LIN {X 0,Y 420.571,Z 343.007,A -85,B 0,C 180,E1 -10184.764,E2 -10184.764} C_VEL
LIN {X 0,Y 421.364,Z 331.747,A -85,B 0,C 180,E1 -10185.601,E2 -10185.601} C_VEL
LIN {X 0,Y 422.031,Z 320.369,A -85,B 0,C 180,E1 -10186.258,E2 -10186.258} C_VEL
LIN {X 0,Y 422.669,Z 307.508,A -85,B 0,C 180,E1 -10186.792,E2 -10186.792} C_VEL
LIN {X 0,Y 423.083,Z 294.135,A -85,B 0,C 180,E1 -10187.148,E2 -10187.148} C_VEL
LIN {X 0,Y 424.009,Z 215.37,A -85,B 0,C 180,E1 -10188.601,E2 -10188.601} C_VEL
LIN {X 0,Y 420.22,Z 192.517,A -85,B 0,C 180,E1 -10189.238,E2 -10189.238} C_VEL
LIN {X 0,Y 419.835,Z 190.333,A -85,B 0,C 180,E1 -10189.315,E2 -10189.315} C_VEL
LIN {X 0,Y 420.887,Z 173.807,A -85,B 0,C 180,E1 -10192.585,E2 -10192.585} C_VEL
LIN {X 0,Y 421.24,Z 166.164,A -85,B 0,C 180,E1 -10194.126,E2 -10194.126} C_VEL
LIN {X 0,Y 418.93,Z 154.675,A -85,B 0,C 180,E1 -10196.664,E2 -10196.664} C_VEL
LIN {X 0,Y 418.192,Z 151.4,A -85,B 0,C 180,E1 -10197.451,E2 -10197.451} C_VEL
LIN {X 0,Y 418.233,Z 151.395,A -85,B 0,C 180,E1 -10200.272,E2 -10200.272} C_VEL
LIN {X 0,Y 418.229,Z 151.389,A -85,B 0,C 180,E1 -10203.678,E2 -10203.678} C_VEL
LIN {X 0,Y 418.231,Z 151.392,A -85,B 0,C 180,E1 -10207.224,E2 -10207.224} C_VEL
LIN {X 0,Y 418.204,Z 151.395,A -85,B 0,C 180,E1 -10210.866,E2 -10210.866} C_VEL
LIN {X 0,Y 418.199,Z 151.393,A -85,B 0,C 180,E1 -10213.727,E2 -10213.727} C_VEL
LIN {X 0,Y 418.195,Z 151.394,A -85,B 0,C 180,E1 -10216.446,E2 -10216.446} C_VEL
LIN {X 0,Y 418.203,Z 151.392,A -85,B 0,C 180,E1 -10219.132,E2 -10219.132} C_VEL
LIN {X 0,Y 418.229,Z 151.388,A -85,B 0,C 180,E1 -10222.774,E2 -10222.774} C_VEL
LIN {X 0,Y 418.226,Z 151.387,A -85,B 0,C 180,E1 -10226.32,E2 -10226.32} C_VEL
LIN {X 0,Y 418.228,Z 151.383,A -85,B 0,C 180,E1 -10229.726,E2 -10229.726} C_VEL
LIN {X 0,Y 418.202,Z 151.386,A -85,B 0,C 180,E1 -10233.016,E2 -10233.016} C_VEL
LIN {X 0,Y 418.248,Z 151.388,A -85,B 0,C 180,E1 -10236.216,E2 -10236.216} C_VEL
LIN {X 0,Y 418.229,Z 151.386,A -85,B 0,C 180,E1 -10239.336,E2 -10239.336} C_VEL
LIN {X 0,Y 418.23,Z 151.389,A -85,B 0,C 180,E1 -10242.393,E2 -10242.393} C_VEL
LIN {X 0,Y 418.268,Z 151.378,A -85,B 0,C 180,E1 -10245.401,E2 -10245.401} C_VEL
LIN {X 0,Y 418.295,Z 151.377,A -85,B 0,C 180,E1 -10248.368,E2 -10248.368} C_VEL
LIN {X 0,Y 418.439,Z 151.361,A -85,B 0,C 180,E1 -10252.278,E2 -10252.278} C_VEL
LIN {X 0,Y 418.461,Z 151.358,A -85,B 0,C 180,E1 -10254.216,E2 -10254.216} C_VEL
LIN {X 0,Y 418.525,Z 151.351,A -85,B 0,C 180,E1 -10258.075,E2 -10258.075} C_VEL
LIN {X 0,Y 418.398,Z 151.362,A -85,B 0,C 180,E1 -10260.962,E2 -10260.962} C_VEL
LIN {X 0,Y 418.46,Z 151.357,A -85,B 0,C 180,E1 -10262.888,E2 -10262.888} C_VEL
LIN {X 0,Y 418.432,Z 151.362,A -85,B 0,C 180,E1 -10266.752,E2 -10266.752} C_VEL
LIN {X 0,Y 418.313,Z 151.381,A -85,B 0,C 180,E1 -10269.672,E2 -10269.672} C_VEL
LIN {X 0,Y 418.338,Z 151.379,A -85,B 0,C 180,E1 -10273,E2 -10273} C_VEL
LIN {X 0,Y 418.251,Z 151.388,A -85,B 0,C 180,E1 -10276.71,E2 -10276.71} C_VEL
LIN {X 0,Y 418.259,Z 151.388,A -85,B 0,C 180,E1 -10280.165,E2 -10280.165} C_VEL
LIN {X 0,Y 418.281,Z 151.439,A -85,B 0,C 180,E1 -10280.537,E2 -10280.537} C_VEL
LIN {X 0,Y 420.491,Z 162.689,A -85,B 0,C 180,E1 -10283.184,E2 -10283.184} C_VEL
LIN {X 0,Y 420.261,Z 170.089,A -85,B 0,C 180,E1 -10284.776,E2 -10284.776} C_VEL
LIN {X 0,Y 424.452,Z 189.753,A -85,B 0,C 180,E1 -10285.38,E2 -10285.38} C_VEL
LIN {X 0,Y 423.071,Z 278.399,A -85,B 0,C 180,E1 -10287.032,E2 -10287.032} C_VEL
LIN {X 0,Y 422.599,Z 291.851,A -85,B 0,C 180,E1 -10287.483,E2 -10287.483} C_VEL
LIN {X 0,Y 422.146,Z 303.797,A -85,B 0,C 180,E1 -10288.074,E2 -10288.074} C_VEL
LIN {X 0,Y 421.53,Z 314.904,A -85,B 0,C 180,E1 -10288.802,E2 -10288.802} C_VEL
LIN {X 0,Y 420.809,Z 325.924,A -85,B 0,C 180,E1 -10289.722,E2 -10289.722} C_VEL
LIN {X 0,Y 420.053,Z 336.491,A -85,B 0,C 180,E1 -10290.823,E2 -10290.823} C_VEL
LIN {X 0,Y 419.339,Z 345.705,A -85,B 0,C 180,E1 -10292.006,E2 -10292.006} C_VEL
LIN {X 0,Y 418.597,Z 354.791,A -85,B 0,C 180,E1 -10293.46,E2 -10293.46} C_VEL
LIN {X 0,Y 418.121,Z 361.803,A -85,B 0,C 180,E1 -10294.854,E2 -10294.854} C_VEL
LIN {X 0,Y 417.75,Z 367.093,A -85,B 0,C 180,E1 -10296.147,E2 -10296.147} C_VEL
LIN {X 0,Y 417.463,Z 372.148,A -85,B 0,C 180,E1 -10297.699,E2 -10297.699} C_VEL
LIN {X 0,Y 417.19,Z 375.839,A -85,B 0,C 180,E1 -10299.204,E2 -10299.204} C_VEL
LIN {X 0,Y 416.986,Z 378.927,A -85,B 0,C 180,E1 -10301.095,E2 -10301.095} C_VEL
LIN {X 0,Y 416.87,Z 380.157,A -85,B 0,C 180,E1 -10302.404,E2 -10302.404} C_VEL
LIN {X 0,Y 416.855,Z 380.606,A -85,B 0,C 180,E1 -10303.728,E2 -10303.728} C_VEL
LIN {X 0,Y 416.898,Z 380.294,A -85,B 0,C 180,E1 -10305.074,E2 -10305.074} C_VEL
LIN {X 0,Y 416.93,Z 379.175,A -85,B 0,C 180,E1 -10306.454,E2 -10306.454} C_VEL
LIN {X 0,Y 417.024,Z 377.173,A -85,B 0,C 180,E1 -10307.86,E2 -10307.86} C_VEL
LIN {X 0,Y 417.209,Z 374.191,A -85,B 0,C 180,E1 -10309.291,E2 -10309.291} C_VEL
LIN {X 0,Y 417.417,Z 370.056,A -85,B 0,C 180,E1 -10310.759,E2 -10310.759} C_VEL
LIN {X 0,Y 417.738,Z 364.602,A -85,B 0,C 180,E1 -10312.253,E2 -10312.253} C_VEL
LIN {X 0,Y 418.142,Z 357.548,A -85,B 0,C 180,E1 -10313.781,E2 -10313.781} C_VEL
LIN {X 0,Y 418.699,Z 349.368,A -85,B 0,C 180,E1 -10315.202,E2 -10315.202} C_VEL
LIN {X 0,Y 419.339,Z 340.676,A -85,B 0,C 180,E1 -10316.423,E2 -10316.423} C_VEL
LIN {X 0,Y 420.009,Z 330.101,A -85,B 0,C 180,E1 -10317.626,E2 -10317.626} C_VEL
LIN {X 0,Y 420.68,Z 318.982,A -85,B 0,C 180,E1 -10318.64,E2 -10318.64} C_VEL
LIN {X 0,Y 421.334,Z 307.001,A -85,B 0,C 180,E1 -10319.489,E2 -10319.489} C_VEL
LIN {X 0,Y 421.864,Z 294.615,A -85,B 0,C 180,E1 -10320.153,E2 -10320.153} C_VEL
LIN {X 0,Y 422.251,Z 281.602,A -85,B 0,C 180,E1 -10320.646,E2 -10320.646} C_VEL
LIN {X 0,Y 422.49,Z 266.058,A -85,B 0,C 180,E1 -10320.988,E2 -10320.988} C_VEL
LIN {X 0,Y 423.528,Z 189.194,A -85,B 0,C 180,E1 -10322.371,E2 -10322.371} C_VEL
LIN {X 0,Y 419.842,Z 169.494,A -85,B 0,C 180,E1 -10322.926,E2 -10322.926} C_VEL
LIN {X 0,Y 420.197,Z 162.178,A -85,B 0,C 180,E1 -10324.578,E2 -10324.578} C_VEL
LIN {X 0,Y 419.152,Z 156.176,A -85,B 0,C 180,E1 -10326.018,E2 -10326.018} C_VEL
LIN {X 0,Y 418.154,Z 154.508,A -85,B 0,C 180,E1 -10326.497,E2 -10326.497} C_VEL
LIN {X 0,Y 416.324,Z 153.399,A -85,B 0,C 180,E1 -10326.973,E2 -10326.973} C_VEL
LIN {X 0,Y 412.363,Z 152.396,A -85,B 0,C 180,E1 -10327.956,E2 -10327.956} C_VEL
LIN {X 0,Y 411.2,Z 152.268,A -85,B 0,C 180,E1 -10328.589,E2 -10328.589} C_VEL
LIN {X 0,Y 411.179,Z 152.266,A -85,B 0,C 180,E1 -10328.683,E2 -10328.683} C_VEL
LIN {X 0,Y 411.209,Z 152.262,A -85,B 0,C 180,E1 -10332.083,E2 -10332.083} C_VEL
LIN {X 0,Y 411.227,Z 152.257,A -85,B 0,C 180,E1 -10335.147,E2 -10335.147} C_VEL
LIN {X 0,Y 411.27,Z 152.256,A -85,B 0,C 180,E1 -10338.167,E2 -10338.167} C_VEL
LIN {X 0,Y 411.384,Z 152.243,A -85,B 0,C 180,E1 -10342.145,E2 -10342.145} C_VEL
LIN {X 0,Y 411.424,Z 152.238,A -85,B 0,C 180,E1 -10344.118,E2 -10344.118} C_VEL
LIN {X 0,Y 411.498,Z 152.229,A -85,B 0,C 180,E1 -10348.043,E2 -10348.043} C_VEL
LIN {X 0,Y 411.373,Z 152.239,A -85,B 0,C 180,E1 -10350.979,E2 -10350.979} C_VEL
LIN {X 0,Y 411.423,Z 152.232,A -85,B 0,C 180,E1 -10352.938,E2 -10352.938} C_VEL
LIN {X 0,Y 411.386,Z 152.237,A -85,B 0,C 180,E1 -10356.868,E2 -10356.868} C_VEL
LIN {X 0,Y 411.272,Z 152.258,A -85,B 0,C 180,E1 -10359.839,E2 -10359.839} C_VEL
LIN {X 0,Y 411.302,Z 152.248,A -85,B 0,C 180,E1 -10363.103,E2 -10363.103} C_VEL
LIN {X 0,Y 411.203,Z 152.26,A -85,B 0,C 180,E1 -10366.891,E2 -10366.891} C_VEL
LIN {X 0,Y 411.2,Z 152.263,A -85,B 0,C 180,E1 -10369.988,E2 -10369.988} C_VEL
LIN {X 0,Y 411.182,Z 152.265,A -85,B 0,C 180,E1 -10373.149,E2 -10373.149} C_VEL
LIN {X 0,Y 411.166,Z 152.264,A -85,B 0,C 180,E1 -10376.386,E2 -10376.386} C_VEL
LIN {X 0,Y 411.188,Z 152.265,A -85,B 0,C 180,E1 -10379.713,E2 -10379.713} C_VEL
LIN {X 0,Y 411.199,Z 152.265,A -85,B 0,C 180,E1 -10383.156,E2 -10383.156} C_VEL
LIN {X 0,Y 411.186,Z 152.262,A -85,B 0,C 180,E1 -10386.552,E2 -10386.552} C_VEL
LIN {X 0,Y 411.163,Z 152.266,A -85,B 0,C 180,E1 -10389.72,E2 -10389.72} C_VEL
LIN {X 0,Y 411.157,Z 152.273,A -85,B 0,C 180,E1 -10393.135,E2 -10393.135} C_VEL
LIN {X 0,Y 411.158,Z 152.266,A -85,B 0,C 180,E1 -10395.882,E2 -10395.882} C_VEL
LIN {X 0,Y 411.152,Z 152.268,A -85,B 0,C 180,E1 -10399.493,E2 -10399.493} C_VEL
LIN {X 0,Y 411.175,Z 152.263,A -85,B 0,C 180,E1 -10402.025,E2 -10402.025} C_VEL
LIN {X 0,Y 411.195,Z 152.265,A -85,B 0,C 180,E1 -10405.124,E2 -10405.124} C_VEL
LIN {X 0,Y 411.157,Z 152.266,A -85,B 0,C 180,E1 -10408.003,E2 -10408.003} C_VEL
LIN {X 0,Y 411.165,Z 152.265,A -85,B 0,C 180,E1 -10411.406,E2 -10411.406} C_VEL
LIN {X 0,Y 411.182,Z 152.266,A -85,B 0,C 180,E1 -10414.941,E2 -10414.941} C_VEL
LIN {X 0,Y 411.194,Z 152.262,A -85,B 0,C 180,E1 -10417.913,E2 -10417.913} C_VEL
LIN {X 0,Y 411.208,Z 152.261,A -85,B 0,C 180,E1 -10421.051,E2 -10421.051} C_VEL
LIN {X 0,Y 411.205,Z 152.263,A -85,B 0,C 180,E1 -10424.13,E2 -10424.13} C_VEL
LIN {X 0,Y 411.296,Z 152.248,A -85,B 0,C 180,E1 -10427.166,E2 -10427.166} C_VEL
LIN {X 0,Y 411.268,Z 152.257,A -85,B 0,C 180,E1 -10430.161,E2 -10430.161} C_VEL
LIN {X 0,Y 411.384,Z 152.237,A -85,B 0,C 180,E1 -10433.132,E2 -10433.132} C_VEL
LIN {X 0,Y 411.278,Z 152.25,A -85,B 0,C 180,E1 -10435.099,E2 -10435.099} C_VEL
LIN {X 0,Y 411.496,Z 152.23,A -85,B 0,C 180,E1 -10438.043,E2 -10438.043} C_VEL
LIN {X 0,Y 411.371,Z 152.239,A -85,B 0,C 180,E1 -10440.979,E2 -10440.979} C_VEL
LIN {X 0,Y 411.42,Z 152.233,A -85,B 0,C 180,E1 -10442.938,E2 -10442.938} C_VEL
LIN {X 0,Y 411.384,Z 152.237,A -85,B 0,C 180,E1 -10446.869,E2 -10446.869} C_VEL
LIN {X 0,Y 411.27,Z 152.259,A -85,B 0,C 180,E1 -10449.84,E2 -10449.84} C_VEL
LIN {X 0,Y 411.301,Z 152.248,A -85,B 0,C 180,E1 -10453.104,E2 -10453.104} C_VEL
LIN {X 0,Y 411.203,Z 152.26,A -85,B 0,C 180,E1 -10456.891,E2 -10456.891} C_VEL
LIN {X 0,Y 411.2,Z 152.263,A -85,B 0,C 180,E1 -10459.989,E2 -10459.989} C_VEL
LIN {X 0,Y 411.182,Z 152.265,A -85,B 0,C 180,E1 -10463.149,E2 -10463.149} C_VEL
LIN {X 0,Y 411.167,Z 152.264,A -85,B 0,C 180,E1 -10466.386,E2 -10466.386} C_VEL
LIN {X 0,Y 411.189,Z 152.265,A -85,B 0,C 180,E1 -10469.714,E2 -10469.714} C_VEL
LIN {X 0,Y 411.201,Z 152.265,A -85,B 0,C 180,E1 -10473.157,E2 -10473.157} C_VEL
LIN {X 0,Y 411.186,Z 152.263,A -85,B 0,C 180,E1 -10476.552,E2 -10476.552} C_VEL
LIN {X 0,Y 411.166,Z 152.266,A -85,B 0,C 180,E1 -10479.721,E2 -10479.721} C_VEL
LIN {X 0,Y 411.159,Z 152.272,A -85,B 0,C 180,E1 -10483.136,E2 -10483.136} C_VEL
LIN {X 0,Y 411.162,Z 152.265,A -85,B 0,C 180,E1 -10485.882,E2 -10485.882} C_VEL
LIN {X 0,Y 411.157,Z 152.267,A -85,B 0,C 180,E1 -10489.493,E2 -10489.493} C_VEL
LIN {X 0,Y 411.18,Z 152.263,A -85,B 0,C 180,E1 -10492.025,E2 -10492.025} C_VEL
LIN {X 0,Y 411.201,Z 152.264,A -85,B 0,C 180,E1 -10495.124,E2 -10495.124} C_VEL
LIN {X 0,Y 411.158,Z 152.266,A -85,B 0,C 180,E1 -10498.002,E2 -10498.002} C_VEL
LIN {X 0,Y 411.169,Z 152.267,A -85,B 0,C 180,E1 -10501.407,E2 -10501.407} C_VEL
LIN {X 0,Y 411.198,Z 152.412,A -85,B 0,C 180,E1 -10502.635,E2 -10502.635} C_VEL
LIN {X 0,Y 413.704,Z 164.762,A -85,B 0,C 180,E1 -10505.405,E2 -10505.405} C_VEL
LIN {X 0,Y 414.113,Z 168.81,A -85,B 0,C 180,E1 -10506.273,E2 -10506.273} C_VEL
LIN {X 0,Y 412.889,Z 187.598,A -85,B 0,C 180,E1 -10510.097,E2 -10510.097} C_VEL
LIN {X 0,Y 412.57,Z 191.176,A -85,B 0,C 180,E1 -10510.815,E2 -10510.815} C_VEL
LIN {X 0,Y 416.564,Z 216.973,A -85,B 0,C 180,E1 -10511.482,E2 -10511.482} C_VEL
LIN {X 0,Y 415.425,Z 299,A -85,B 0,C 180,E1 -10513.001,E2 -10513.001} C_VEL
LIN {X 0,Y 414.972,Z 312.17,A -85,B 0,C 180,E1 -10513.425,E2 -10513.425} C_VEL
LIN {X 0,Y 414.389,Z 324.339,A -85,B 0,C 180,E1 -10514.002,E2 -10514.002} C_VEL
LIN {X 0,Y 413.724,Z 335.853,A -85,B 0,C 180,E1 -10514.734,E2 -10514.734} C_VEL
LIN {X 0,Y 413.008,Z 346.776,A -85,B 0,C 180,E1 -10515.627,E2 -10515.627} C_VEL
LIN {X 0,Y 412.258,Z 358.362,A -85,B 0,C 180,E1 -10516.826,E2 -10516.826} C_VEL
LIN {X 0,Y 411.689,Z 366.989,A -85,B 0,C 180,E1 -10517.929,E2 -10517.929} C_VEL
LIN {X 0,Y 411.068,Z 374.981,A -85,B 0,C 180,E1 -10519.16,E2 -10519.16} C_VEL
LIN {X 0,Y 410.605,Z 382.783,A -85,B 0,C 180,E1 -10520.642,E2 -10520.642} C_VEL
LIN {X 0,Y 410.285,Z 389.031,A -85,B 0,C 180,E1 -10522.124,E2 -10522.124} C_VEL
LIN {X 0,Y 410.071,Z 394.382,A -85,B 0,C 180,E1 -10523.741,E2 -10523.741} C_VEL
LIN {X 0,Y 410.016,Z 397.784,A -85,B 0,C 180,E1 -10525.083,E2 -10525.083} C_VEL
LIN {X 0,Y 409.932,Z 399.737,A -85,B 0,C 180,E1 -10526.068,E2 -10526.068} C_VEL
LIN {X 0,Y 409.927,Z 401.26,A -85,B 0,C 180,E1 -10527.052,E2 -10527.052} C_VEL
LIN {X 0,Y 409.967,Z 402.321,A -85,B 0,C 180,E1 -10528.035,E2 -10528.035} C_VEL
LIN {X 0,Y 409.937,Z 402.979,A -85,B 0,C 180,E1 -10529.018,E2 -10529.018} C_VEL
LIN {X 0,Y 409.928,Z 403.244,A -85,B 0,C 180,E1 -10530,E2 -10530} C_VEL
LIN {X 0,Y 409.937,Z 403.101,A -85,B 0,C 180,E1 -10530.982,E2 -10530.982} C_VEL
LIN {X 0,Y 409.967,Z 402.517,A -85,B 0,C 180,E1 -10531.965,E2 -10531.965} C_VEL
LIN {X 0,Y 409.925,Z 401.535,A -85,B 0,C 180,E1 -10532.948,E2 -10532.948} C_VEL
LIN {X 0,Y 409.931,Z 400.152,A -85,B 0,C 180,E1 -10533.932,E2 -10533.932} C_VEL
LIN {X 0,Y 410.012,Z 397.234,A -85,B 0,C 180,E1 -10535.409,E2 -10535.409} C_VEL
LIN {X 0,Y 410.168,Z 393.27,A -85,B 0,C 180,E1 -10536.888,E2 -10536.888} C_VEL
LIN {X 0,Y 410.475,Z 387.186,A -85,B 0,C 180,E1 -10538.616,E2 -10538.616} C_VEL
LIN {X 0,Y 410.914,Z 380.501,A -85,B 0,C 180,E1 -10540.096,E2 -10540.096} C_VEL
LIN {X 0,Y 411.512,Z 372.217,A -85,B 0,C 180,E1 -10541.576,E2 -10541.576} C_VEL
LIN {X 0,Y 412.276,Z 363.768,A -85,B 0,C 180,E1 -10542.803,E2 -10542.803} C_VEL
LIN {X 0,Y 412.884,Z 354.377,A -85,B 0,C 180,E1 -10543.93,E2 -10543.93} C_VEL
LIN {X 0,Y 413.697,Z 343.103,A -85,B 0,C 180,E1 -10545.015,E2 -10545.015} C_VEL
LIN {X 0,Y 414.549,Z 331.915,A -85,B 0,C 180,E1 -10545.865,E2 -10545.865} C_VEL
LIN {X 0,Y 415.239,Z 320.652,A -85,B 0,C 180,E1 -10546.532,E2 -10546.532} C_VEL
LIN {X 0,Y 415.858,Z 308.078,A -85,B 0,C 180,E1 -10547.075,E2 -10547.075} C_VEL
LIN {X 0,Y 416.322,Z 295.194,A -85,B 0,C 180,E1 -10547.436,E2 -10547.436} C_VEL
LIN {X 0,Y 417.379,Z 216.328,A -85,B 0,C 180,E1 -10548.919,E2 -10548.919} C_VEL
LIN {X 0,Y 413.666,Z 194.049,A -85,B 0,C 180,E1 -10549.561,E2 -10549.561} C_VEL
LIN {X 0,Y 412.977,Z 190.144,A -85,B 0,C 180,E1 -10549.685,E2 -10549.685} C_VEL
LIN {X 0,Y 414.183,Z 172.189,A -85,B 0,C 180,E1 -10553.309,E2 -10553.309} C_VEL
LIN {X 0,Y 414.313,Z 167.438,A -85,B 0,C 180,E1 -10554.289,E2 -10554.289} C_VEL
LIN {X 0,Y 411.997,Z 156.051,A -85,B 0,C 180,E1 -10556.865,E2 -10556.865} C_VEL
LIN {X 0,Y 411.173,Z 152.274,A -85,B 0,C 180,E1 -10557.76,E2 -10557.76} C_VEL
LIN {X 0,Y 411.182,Z 152.274,A -85,B 0,C 180,E1 -10560.848,E2 -10560.848} C_VEL
LIN {X 0,Y 411.19,Z 152.265,A -85,B 0,C 180,E1 -10564.334,E2 -10564.334} C_VEL
LIN {X 0,Y 411.183,Z 152.268,A -85,B 0,C 180,E1 -10566.742,E2 -10566.742} C_VEL
LIN {X 0,Y 411.165,Z 152.27,A -85,B 0,C 180,E1 -10569.719,E2 -10569.719} C_VEL
LIN {X 0,Y 411.159,Z 152.273,A -85,B 0,C 180,E1 -10573.134,E2 -10573.134} C_VEL
LIN {X 0,Y 411.159,Z 152.268,A -85,B 0,C 180,E1 -10575.881,E2 -10575.881} C_VEL
LIN {X 0,Y 411.154,Z 152.267,A -85,B 0,C 180,E1 -10579.492,E2 -10579.492} C_VEL
LIN {X 0,Y 411.177,Z 152.265,A -85,B 0,C 180,E1 -10582.024,E2 -10582.024} C_VEL
LIN {X 0,Y 411.197,Z 152.264,A -85,B 0,C 180,E1 -10585.123,E2 -10585.123} C_VEL
LIN {X 0,Y 411.154,Z 152.267,A -85,B 0,C 180,E1 -10588.001,E2 -10588.001} C_VEL
LIN {X 0,Y 411.163,Z 152.266,A -85,B 0,C 180,E1 -10591.405,E2 -10591.405} C_VEL
LIN {X 0,Y 411.182,Z 152.266,A -85,B 0,C 180,E1 -10594.941,E2 -10594.941} C_VEL
LIN {X 0,Y 411.192,Z 152.258,A -85,B 0,C 180,E1 -10597.912,E2 -10597.912} C_VEL
LIN {X 0,Y 411.176,Z 152.26,A -85,B 0,C 180,E1 -10601.049,E2 -10601.049} C_VEL
LIN {X 0,Y 411.201,Z 152.263,A -85,B 0,C 180,E1 -10604.129,E2 -10604.129} C_VEL
LIN {X 0,Y 411.295,Z 152.249,A -85,B 0,C 180,E1 -10607.165,E2 -10607.165} C_VEL
LIN {X 0,Y 411.268,Z 152.259,A -85,B 0,C 180,E1 -10610.16,E2 -10610.16} C_VEL
LIN {X 0,Y 411.382,Z 152.239,A -85,B 0,C 180,E1 -10613.131,E2 -10613.131} C_VEL
LIN {X 0,Y 411.276,Z 152.248,A -85,B 0,C 180,E1 -10615.098,E2 -10615.098} C_VEL
LIN {X 0,Y 411.494,Z 152.227,A -85,B 0,C 180,E1 -10618.042,E2 -10618.042} C_VEL
LIN {X 0,Y 411.368,Z 152.238,A -85,B 0,C 180,E1 -10620.978,E2 -10620.978} C_VEL
LIN {X 0,Y 411.419,Z 152.235,A -85,B 0,C 180,E1 -10622.937,E2 -10622.937} C_VEL
LIN {X 0,Y 411.382,Z 152.24,A -85,B 0,C 180,E1 -10626.868,E2 -10626.868} C_VEL
LIN {X 0,Y 411.267,Z 152.26,A -85,B 0,C 180,E1 -10629.839,E2 -10629.839} C_VEL
LIN {X 0,Y 411.297,Z 152.257,A -85,B 0,C 180,E1 -10633.103,E2 -10633.103} C_VEL
LIN {X 0,Y 411.2,Z 152.267,A -85,B 0,C 180,E1 -10636.891,E2 -10636.891} C_VEL
LIN {X 0,Y 411.234,Z 152.347,A -85,B 0,C 180,E1 -10640.214,E2 -10640.214} C_VEL
LIN {X 0,Y 413.559,Z 163.936,A -85,B 0,C 180,E1 -10643.008,E2 -10643.008} C_VEL
LIN {X 0,Y 413.416,Z 170.133,A -85,B 0,C 180,E1 -10644.379,E2 -10644.379} C_VEL
LIN {X 0,Y 417.825,Z 190.845,A -85,B 0,C 180,E1 -10645.057,E2 -10645.057} C_VEL
LIN {X 0,Y 416.347,Z 278.62,A -85,B 0,C 180,E1 -10646.721,E2 -10646.721} C_VEL
LIN {X 0,Y 415.857,Z 292.111,A -85,B 0,C 180,E1 -10647.182,E2 -10647.182} C_VEL
LIN {X 0,Y 415.375,Z 304.284,A -85,B 0,C 180,E1 -10647.797,E2 -10647.797} C_VEL
LIN {X 0,Y 414.637,Z 316.272,A -85,B 0,C 180,E1 -10648.609,E2 -10648.609} C_VEL
LIN {X 0,Y 413.835,Z 327.728,A -85,B 0,C 180,E1 -10649.605,E2 -10649.605} C_VEL
LIN {X 0,Y 413.103,Z 337.69,A -85,B 0,C 180,E1 -10650.689,E2 -10650.689} C_VEL
LIN {X 0,Y 412.349,Z 346.691,A -85,B 0,C 180,E1 -10651.894,E2 -10651.894} C_VEL
LIN {X 0,Y 411.561,Z 355.998,A -85,B 0,C 180,E1 -10653.44,E2 -10653.44} C_VEL
LIN {X 0,Y 411.062,Z 362.796,A -85,B 0,C 180,E1 -10654.85,E2 -10654.85} C_VEL
LIN {X 0,Y 410.606,Z 368.893,A -85,B 0,C 180,E1 -10656.443,E2 -10656.443} C_VEL
LIN {X 0,Y 410.3,Z 373.675,A -85,B 0,C 180,E1 -10658.071,E2 -10658.071} C_VEL
LIN {X 0,Y 410.05,Z 376.872,A -85,B 0,C 180,E1 -10659.533,E2 -10659.533} C_VEL
LIN {X 0,Y 409.897,Z 379.134,A -85,B 0,C 180,E1 -10661.027,E2 -10661.027} C_VEL
LIN {X 0,Y 409.778,Z 380.421,A -85,B 0,C 180,E1 -10662.484,E2 -10662.484} C_VEL
LIN {X 0,Y 409.765,Z 380.823,A -85,B 0,C 180,E1 -10663.917,E2 -10663.917} C_VEL
LIN {X 0,Y 409.801,Z 380.359,A -85,B 0,C 180,E1 -10665.322,E2 -10665.322} C_VEL
LIN {X 0,Y 409.859,Z 379.105,A -85,B 0,C 180,E1 -10666.695,E2 -10666.695} C_VEL
LIN {X 0,Y 409.942,Z 377.104,A -85,B 0,C 180,E1 -10668.041,E2 -10668.041} C_VEL
LIN {X 0,Y 410.123,Z 374.338,A -85,B 0,C 180,E1 -10669.37,E2 -10669.37} C_VEL
LIN {X 0,Y 410.378,Z 369.74,A -85,B 0,C 180,E1 -10670.998,E2 -10670.998} C_VEL
LIN {X 0,Y 410.763,Z 363.813,A -85,B 0,C 180,E1 -10672.6,E2 -10672.6} C_VEL
LIN {X 0,Y 411.131,Z 357.385,A -85,B 0,C 180,E1 -10673.986,E2 -10673.986} C_VEL
LIN {X 0,Y 411.698,Z 349.368,A -85,B 0,C 180,E1 -10675.391,E2 -10675.391} C_VEL
LIN {X 0,Y 412.361,Z 340.662,A -85,B 0,C 180,E1 -10676.628,E2 -10676.628} C_VEL
LIN {X 0,Y 413.079,Z 329.742,A -85,B 0,C 180,E1 -10677.882,E2 -10677.882} C_VEL
LIN {X 0,Y 413.731,Z 319.858,A -85,B 0,C 180,E1 -10678.796,E2 -10678.796} C_VEL
LIN {X 0,Y 414.372,Z 308.144,A -85,B 0,C 180,E1 -10679.66,E2 -10679.66} C_VEL
LIN {X 0,Y 414.949,Z 295.958,A -85,B 0,C 180,E1 -10680.338,E2 -10680.338} C_VEL
LIN {X 0,Y 415.323,Z 283.209,A -85,B 0,C 180,E1 -10680.848,E2 -10680.848} C_VEL
LIN {X 0,Y 415.646,Z 270.271,A -85,B 0,C 180,E1 -10681.167,E2 -10681.167} C_VEL
LIN {X 0,Y 416.691,Z 189.774,A -85,B 0,C 180,E1 -10682.645,E2 -10682.645} C_VEL
LIN {X 0,Y 412.925,Z 169.861,A -85,B 0,C 180,E1 -10683.191,E2 -10683.191} C_VEL
LIN {X 0,Y 413.153,Z 162.681,A -85,B 0,C 180,E1 -10684.833,E2 -10684.833} C_VEL
LIN {X 0,Y 411.195,Z 152.266,A -85,B 0,C 180,E1 -10687.411,E2 -10687.411} C_VEL
LIN {X 0,Y 411.179,Z 152.266,A -85,B 0,C 180,E1 -10688.683,E2 -10688.683} C_VEL
LIN {X 0,Y 410.533,Z 152.35,A -85,B 0,C 180,E1 -10689.5,E2 -10689.5} C_VEL
LIN {X 0,Y 407.698,Z 152.706,A -85,B 0,C 180,E1 -10690.829,E2 -10690.829} C_VEL
LIN {X 0,Y 405.288,Z 153.004,A -85,B 0,C 180,E1 -10691.902,E2 -10691.902} C_VEL
LIN {X 0,Y 404.253,Z 153.13,A -85,B 0,C 180,E1 -10692.731,E2 -10692.731} C_VEL
LIN {X 0,Y 404.17,Z 153.137,A -85,B 0,C 180,E1 -10693.012,E2 -10693.012} C_VEL
LIN {X 0,Y 404.28,Z 153.124,A -85,B 0,C 180,E1 -10696.939,E2 -10696.939} C_VEL
LIN {X 0,Y 404.239,Z 153.131,A -85,B 0,C 180,E1 -10699.988,E2 -10699.988} C_VEL
LIN {X 0,Y 404.336,Z 153.116,A -85,B 0,C 180,E1 -10703.012,E2 -10703.012} C_VEL
LIN {X 0,Y 404.255,Z 153.126,A -85,B 0,C 180,E1 -10705.013,E2 -10705.013} C_VEL
LIN {X 0,Y 404.467,Z 153.104,A -85,B 0,C 180,E1 -10708.009,E2 -10708.009} C_VEL
LIN {X 0,Y 404.344,Z 153.114,A -85,B 0,C 180,E1 -10710.996,E2 -10710.996} C_VEL
LIN {X 0,Y 404.356,Z 153.113,A -85,B 0,C 180,E1 -10712.989,E2 -10712.989} C_VEL
LIN {X 0,Y 404.363,Z 153.119,A -85,B 0,C 180,E1 -10715.986,E2 -10715.986} C_VEL
LIN {X 0,Y 404.252,Z 153.126,A -85,B 0,C 180,E1 -10719.002,E2 -10719.002} C_VEL
LIN {X 0,Y 404.245,Z 153.131,A -85,B 0,C 180,E1 -10722.042,E2 -10722.042} C_VEL
LIN {X 0,Y 404.17,Z 153.137,A -85,B 0,C 180,E1 -10725.119,E2 -10725.119} C_VEL
LIN {X 0,Y 404.131,Z 153.142,A -85,B 0,C 180,E1 -10728.242,E2 -10728.242} C_VEL
LIN {X 0,Y 404.126,Z 153.146,A -85,B 0,C 180,E1 -10731.42,E2 -10731.42} C_VEL
LIN {X 0,Y 404.131,Z 153.141,A -85,B 0,C 180,E1 -10734.668,E2 -10734.668} C_VEL
LIN {X 0,Y 404.096,Z 153.147,A -85,B 0,C 180,E1 -10738.007,E2 -10738.007} C_VEL
LIN {X 0,Y 404.135,Z 153.14,A -85,B 0,C 180,E1 -10740.286,E2 -10740.286} C_VEL
LIN {X 0,Y 404.133,Z 153.142,A -85,B 0,C 180,E1 -10743.813,E2 -10743.813} C_VEL
LIN {X 0,Y 404.129,Z 153.144,A -85,B 0,C 180,E1 -10746.874,E2 -10746.874} C_VEL
LIN {X 0,Y 404.112,Z 153.143,A -85,B 0,C 180,E1 -10750.075,E2 -10750.075} C_VEL
LIN {X 0,Y 404.136,Z 153.147,A -85,B 0,C 180,E1 -10753.082,E2 -10753.082} C_VEL
LIN {X 0,Y 404.115,Z 153.143,A -85,B 0,C 180,E1 -10755.922,E2 -10755.922} C_VEL
LIN {X 0,Y 404.096,Z 153.148,A -85,B 0,C 180,E1 -10758.633,E2 -10758.633} C_VEL
LIN {X 0,Y 404.132,Z 153.142,A -85,B 0,C 180,E1 -10761.495,E2 -10761.495} C_VEL
LIN {X 0,Y 404.166,Z 153.142,A -85,B 0,C 180,E1 -10764.983,E2 -10764.983} C_VEL
LIN {X 0,Y 404.131,Z 153.144,A -85,B 0,C 180,E1 -10768.443,E2 -10768.443} C_VEL
LIN {X 0,Y 404.143,Z 153.145,A -85,B 0,C 180,E1 -10770.862,E2 -10770.862} C_VEL
LIN {X 0,Y 404.147,Z 153.145,A -85,B 0,C 180,E1 -10774.723,E2 -10774.723} C_VEL
LIN {X 0,Y 404.158,Z 153.137,A -85,B 0,C 180,E1 -10777.508,E2 -10777.508} C_VEL
LIN {X 0,Y 404.153,Z 153.143,A -85,B 0,C 180,E1 -10780.707,E2 -10780.707} C_VEL
LIN {X 0,Y 404.175,Z 153.137,A -85,B 0,C 180,E1 -10783.847,E2 -10783.847} C_VEL
LIN {X 0,Y 404.278,Z 153.124,A -85,B 0,C 180,E1 -10786.939,E2 -10786.939} C_VEL
LIN {X 0,Y 404.236,Z 153.131,A -85,B 0,C 180,E1 -10789.988,E2 -10789.988} C_VEL
LIN {X 0,Y 404.334,Z 153.116,A -85,B 0,C 180,E1 -10793.012,E2 -10793.012} C_VEL
LIN {X 0,Y 404.25,Z 153.126,A -85,B 0,C 180,E1 -10795.014,E2 -10795.014} C_VEL
LIN {X 0,Y 404.465,Z 153.105,A -85,B 0,C 180,E1 -10798.009,E2 -10798.009} C_VEL
LIN {X 0,Y 404.341,Z 153.115,A -85,B 0,C 180,E1 -10800.996,E2 -10800.996} C_VEL
LIN {X 0,Y 404.354,Z 153.113,A -85,B 0,C 180,E1 -10802.989,E2 -10802.989} C_VEL
LIN {X 0,Y 404.361,Z 153.119,A -85,B 0,C 180,E1 -10805.986,E2 -10805.986} C_VEL
LIN {X 0,Y 404.25,Z 153.126,A -85,B 0,C 180,E1 -10809.002,E2 -10809.002} C_VEL
LIN {X 0,Y 404.244,Z 153.131,A -85,B 0,C 180,E1 -10812.042,E2 -10812.042} C_VEL
LIN {X 0,Y 404.169,Z 153.137,A -85,B 0,C 180,E1 -10815.12,E2 -10815.12} C_VEL
LIN {X 0,Y 404.131,Z 153.142,A -85,B 0,C 180,E1 -10818.242,E2 -10818.242} C_VEL
LIN {X 0,Y 404.126,Z 153.147,A -85,B 0,C 180,E1 -10821.42,E2 -10821.42} C_VEL
LIN {X 0,Y 404.131,Z 153.141,A -85,B 0,C 180,E1 -10824.669,E2 -10824.669} C_VEL
LIN {X 0,Y 404.097,Z 153.146,A -85,B 0,C 180,E1 -10828.007,E2 -10828.007} C_VEL
LIN {X 0,Y 404.136,Z 153.14,A -85,B 0,C 180,E1 -10830.286,E2 -10830.286} C_VEL
LIN {X 0,Y 404.135,Z 153.142,A -85,B 0,C 180,E1 -10833.814,E2 -10833.814} C_VEL
LIN {X 0,Y 404.129,Z 153.144,A -85,B 0,C 180,E1 -10836.874,E2 -10836.874} C_VEL
LIN {X 0,Y 404.115,Z 153.143,A -85,B 0,C 180,E1 -10840.075,E2 -10840.075} C_VEL
LIN {X 0,Y 404.139,Z 153.147,A -85,B 0,C 180,E1 -10843.082,E2 -10843.082} C_VEL
LIN {X 0,Y 404.119,Z 153.142,A -85,B 0,C 180,E1 -10845.923,E2 -10845.923} C_VEL
LIN {X 0,Y 404.1,Z 153.148,A -85,B 0,C 180,E1 -10848.633,E2 -10848.633} C_VEL
LIN {X 0,Y 404.137,Z 153.141,A -85,B 0,C 180,E1 -10851.496,E2 -10851.496} C_VEL
LIN {X 0,Y 404.172,Z 153.141,A -85,B 0,C 180,E1 -10854.983,E2 -10854.983} C_VEL
LIN {X 0,Y 404.133,Z 153.144,A -85,B 0,C 180,E1 -10858.444,E2 -10858.444} C_VEL
LIN {X 0,Y 404.147,Z 153.143,A -85,B 0,C 180,E1 -10860.863,E2 -10860.863} C_VEL
LIN {X 0,Y 404.132,Z 153.171,A -85,B 0,C 180,E1 -10862.364,E2 -10862.364} C_VEL
LIN {X 0,Y 406.641,Z 165.679,A -85,B 0,C 180,E1 -10865.222,E2 -10865.222} C_VEL
LIN {X 0,Y 407.148,Z 170.087,A -85,B 0,C 180,E1 -10866.187,E2 -10866.187} C_VEL
LIN {X 0,Y 405.875,Z 188.523,A -85,B 0,C 180,E1 -10870.002,E2 -10870.002} C_VEL
LIN {X 0,Y 405.659,Z 190.888,A -85,B 0,C 180,E1 -10870.486,E2 -10870.486} C_VEL
LIN {X 0,Y 409.741,Z 217.611,A -85,B 0,C 180,E1 -10871.209,E2 -10871.209} C_VEL
LIN {X 0,Y 408.592,Z 298.715,A -85,B 0,C 180,E1 -10872.74,E2 -10872.74} C_VEL
LIN {X 0,Y 408.099,Z 311.906,A -85,B 0,C 180,E1 -10873.17,E2 -10873.17} C_VEL
LIN {X 0,Y 407.489,Z 324.656,A -85,B 0,C 180,E1 -10873.788,E2 -10873.788} C_VEL
LIN {X 0,Y 406.728,Z 336.846,A -85,B 0,C 180,E1 -10874.593,E2 -10874.593} C_VEL
LIN {X 0,Y 405.911,Z 348.438,A -85,B 0,C 180,E1 -10875.588,E2 -10875.588} C_VEL
LIN {X 0,Y 405.215,Z 359.159,A -85,B 0,C 180,E1 -10876.745,E2 -10876.745} C_VEL
LIN {X 0,Y 404.576,Z 368.295,A -85,B 0,C 180,E1 -10877.968,E2 -10877.968} C_VEL
LIN {X 0,Y 403.884,Z 377.387,A -85,B 0,C 180,E1 -10879.472,E2 -10879.472} C_VEL
LIN {X 0,Y 403.454,Z 384.709,A -85,B 0,C 180,E1 -10880.98,E2 -10880.98} C_VEL
LIN {X 0,Y 403.137,Z 390.543,A -85,B 0,C 180,E1 -10882.487,E2 -10882.487} C_VEL
LIN {X 0,Y 402.94,Z 395.119,A -85,B 0,C 180,E1 -10883.993,E2 -10883.993} C_VEL
LIN {X 0,Y 402.928,Z 397.525,A -85,B 0,C 180,E1 -10884.997,E2 -10884.997} C_VEL
LIN {X 0,Y 402.852,Z 399.49,A -85,B 0,C 180,E1 -10885.998,E2 -10885.998} C_VEL
LIN {X 0,Y 402.826,Z 401.028,A -85,B 0,C 180,E1 -10887,E2 -10887} C_VEL
LIN {X 0,Y 402.865,Z 402.103,A -85,B 0,C 180,E1 -10888,E2 -10888} C_VEL
LIN {X 0,Y 402.864,Z 402.771,A -85,B 0,C 180,E1 -10889,E2 -10889} C_VEL
LIN {X 0,Y 402.853,Z 403.044,A -85,B 0,C 180,E1 -10890,E2 -10890} C_VEL
LIN {X 0,Y 402.864,Z 402.914,A -85,B 0,C 180,E1 -10890.999,E2 -10890.999} C_VEL
LIN {X 0,Y 402.865,Z 402.34,A -85,B 0,C 180,E1 -10891.999,E2 -10891.999} C_VEL
LIN {X 0,Y 402.851,Z 399.988,A -85,B 0,C 180,E1 -10894.001,E2 -10894.001} C_VEL
LIN {X 0,Y 402.91,Z 397.082,A -85,B 0,C 180,E1 -10895.505,E2 -10895.505} C_VEL
LIN {X 0,Y 403.081,Z 393.137,A -85,B 0,C 180,E1 -10897.01,E2 -10897.01} C_VEL
LIN {X 0,Y 403.361,Z 388.052,A -85,B 0,C 180,E1 -10898.517,E2 -10898.517} C_VEL
LIN {X 0,Y 403.804,Z 381.67,A -85,B 0,C 180,E1 -10900.023,E2 -10900.023} C_VEL
LIN {X 0,Y 404.386,Z 373.685,A -85,B 0,C 180,E1 -10901.529,E2 -10901.529} C_VEL
LIN {X 0,Y 405.171,Z 365.56,A -85,B 0,C 180,E1 -10902.777,E2 -10902.777} C_VEL
LIN {X 0,Y 405.869,Z 355.666,A -85,B 0,C 180,E1 -10904.029,E2 -10904.029} C_VEL
LIN {X 0,Y 406.753,Z 344.629,A -85,B 0,C 180,E1 -10905.149,E2 -10905.149} C_VEL
LIN {X 0,Y 407.742,Z 332.084,A -85,B 0,C 180,E1 -10906.137,E2 -10906.137} C_VEL
LIN {X 0,Y 408.537,Z 319.782,A -85,B 0,C 180,E1 -10906.875,E2 -10906.875} C_VEL
LIN {X 0,Y 409.217,Z 306.856,A -85,B 0,C 180,E1 -10907.426,E2 -10907.426} C_VEL
LIN {X 0,Y 409.676,Z 293.402,A -85,B 0,C 180,E1 -10907.792,E2 -10907.792} C_VEL
LIN {X 0,Y 410.772,Z 217.27,A -85,B 0,C 180,E1 -10909.25,E2 -10909.25} C_VEL
LIN {X 0,Y 407.043,Z 194.914,A -85,B 0,C 180,E1 -10909.915,E2 -10909.915} C_VEL
LIN {X 0,Y 406.108,Z 189.823,A -85,B 0,C 180,E1 -10910.1,E2 -10910.1} C_VEL
LIN {X 0,Y 407.255,Z 173.821,A -85,B 0,C 180,E1 -10913.385,E2 -10913.385} C_VEL
LIN {X 0,Y 407.385,Z 168.743,A -85,B 0,C 180,E1 -10914.458,E2 -10914.458} C_VEL
LIN {X 0,Y 405.336,Z 158.606,A -85,B 0,C 180,E1 -10916.795,E2 -10916.795} C_VEL
LIN {X 0,Y 404.126,Z 153.15,A -85,B 0,C 180,E1 -10918.145,E2 -10918.145} C_VEL
LIN {X 0,Y 404.132,Z 153.15,A -85,B 0,C 180,E1 -10921.555,E2 -10921.555} C_VEL
LIN {X 0,Y 404.171,Z 153.142,A -85,B 0,C 180,E1 -10925.017,E2 -10925.017} C_VEL
LIN {X 0,Y 404.13,Z 153.147,A -85,B 0,C 180,E1 -10928.759,E2 -10928.759} C_VEL
LIN {X 0,Y 404.104,Z 153.151,A -85,B 0,C 180,E1 -10931.596,E2 -10931.596} C_VEL
LIN {X 0,Y 404.14,Z 153.147,A -85,B 0,C 180,E1 -10934.521,E2 -10934.521} C_VEL
LIN {X 0,Y 404.116,Z 153.144,A -85,B 0,C 180,E1 -10937.292,E2 -10937.292} C_VEL
LIN {X 0,Y 404.129,Z 153.142,A -85,B 0,C 180,E1 -10939.95,E2 -10939.95} C_VEL
LIN {X 0,Y 404.127,Z 153.141,A -85,B 0,C 180,E1 -10943.125,E2 -10943.125} C_VEL
LIN {X 0,Y 404.133,Z 153.143,A -85,B 0,C 180,E1 -10946.186,E2 -10946.186} C_VEL
LIN {X 0,Y 404.134,Z 153.138,A -85,B 0,C 180,E1 -10949.713,E2 -10949.713} C_VEL
LIN {X 0,Y 404.096,Z 153.142,A -85,B 0,C 180,E1 -10953.115,E2 -10953.115} C_VEL
LIN {X 0,Y 404.141,Z 153.142,A -85,B 0,C 180,E1 -10956.423,E2 -10956.423} C_VEL
LIN {X 0,Y 404.144,Z 153.143,A -85,B 0,C 180,E1 -10959.89,E2 -10959.89} C_VEL
LIN {X 0,Y 404.149,Z 153.141,A -85,B 0,C 180,E1 -10963.021,E2 -10963.021} C_VEL
LIN {X 0,Y 404.277,Z 153.124,A -85,B 0,C 180,E1 -10966.938,E2 -10966.938} C_VEL
LIN {X 0,Y 404.236,Z 153.133,A -85,B 0,C 180,E1 -10969.987,E2 -10969.987} C_VEL
LIN {X 0,Y 404.333,Z 153.118,A -85,B 0,C 180,E1 -10973.011,E2 -10973.011} C_VEL
LIN {X 0,Y 404.248,Z 153.123,A -85,B 0,C 180,E1 -10975.013,E2 -10975.013} C_VEL
LIN {X 0,Y 404.462,Z 153.102,A -85,B 0,C 180,E1 -10978.008,E2 -10978.008} C_VEL
LIN {X 0,Y 404.339,Z 153.114,A -85,B 0,C 180,E1 -10980.996,E2 -10980.996} C_VEL
LIN {X 0,Y 404.378,Z 153.112,A -85,B 0,C 180,E1 -10982.988,E2 -10982.988} C_VEL
LIN {X 0,Y 404.332,Z 153.119,A -85,B 0,C 180,E1 -10986.988,E2 -10986.988} C_VEL
LIN {X 0,Y 404.235,Z 153.137,A -85,B 0,C 180,E1 -10990.012,E2 -10990.012} C_VEL
LIN {X 0,Y 404.26,Z 153.134,A -85,B 0,C 180,E1 -10993.211,E2 -10993.211} C_VEL
LIN {X 0,Y 404.169,Z 153.144,A -85,B 0,C 180,E1 -10997.194,E2 -10997.194} C_VEL
LIN {X 0,Y 404.204,Z 153.211,A -85,B 0,C 180,E1 -10999.871,E2 -10999.871} C_VEL
LIN {X 0,Y 406.505,Z 164.355,A -85,B 0,C 180,E1 -11002.623,E2 -11002.623} C_VEL
LIN {X 0,Y 406.628,Z 170.063,A -85,B 0,C 180,E1 -11003.926,E2 -11003.926} C_VEL
LIN {X 0,Y 406.623,Z 170.596,A -85,B 0,C 180,E1 -11004.013,E2 -11004.013} C_VEL
LIN {X 0,Y 411.144,Z 191.428,A -85,B 0,C 180,E1 -11004.701,E2 -11004.701} C_VEL
LIN {X 0,Y 409.648,Z 278.945,A -85,B 0,C 180,E1 -11006.405,E2 -11006.405} C_VEL
LIN {X 0,Y 409.137,Z 292.265,A -85,B 0,C 180,E1 -11006.867,E2 -11006.867} C_VEL
LIN {X 0,Y 408.626,Z 304.358,A -85,B 0,C 180,E1 -11007.486,E2 -11007.486} C_VEL
LIN {X 0,Y 407.874,Z 316.103,A -85,B 0,C 180,E1 -11008.288,E2 -11008.288} C_VEL
LIN {X 0,Y 406.998,Z 328.025,A -85,B 0,C 180,E1 -11009.339,E2 -11009.339} C_VEL
LIN {X 0,Y 406.25,Z 337.625,A -85,B 0,C 180,E1 -11010.398,E2 -11010.398} C_VEL
LIN {X 0,Y 405.514,Z 346.354,A -85,B 0,C 180,E1 -11011.573,E2 -11011.573} C_VEL
LIN {X 0,Y 404.678,Z 355.097,A -85,B 0,C 180,E1 -11013.021,E2 -11013.021} C_VEL
LIN {X 0,Y 404.15,Z 361.903,A -85,B 0,C 180,E1 -11014.413,E2 -11014.413} C_VEL
LIN {X 0,Y 403.66,Z 368.109,A -85,B 0,C 180,E1 -11015.99,E2 -11015.99} C_VEL
LIN {X 0,Y 403.299,Z 372.99,A -85,B 0,C 180,E1 -11017.583,E2 -11017.583} C_VEL
LIN {X 0,Y 403.061,Z 376.021,A -85,B 0,C 180,E1 -11018.881,E2 -11018.881} C_VEL
LIN {X 0,Y 402.887,Z 378.338,A -85,B 0,C 180,E1 -11020.197,E2 -11020.197} C_VEL
LIN {X 0,Y 402.745,Z 379.966,A -85,B 0,C 180,E1 -11021.537,E2 -11021.537} C_VEL
LIN {X 0,Y 402.661,Z 380.836,A -85,B 0,C 180,E1 -11022.898,E2 -11022.898} C_VEL
LIN {X 0,Y 402.681,Z 380.947,A -85,B 0,C 180,E1 -11024.311,E2 -11024.311} C_VEL
LIN {X 0,Y 402.706,Z 380.262,A -85,B 0,C 180,E1 -11025.728,E2 -11025.728} C_VEL
LIN {X 0,Y 402.803,Z 378.804,A -85,B 0,C 180,E1 -11027.121,E2 -11027.121} C_VEL
LIN {X 0,Y 402.911,Z 376.361,A -85,B 0,C 180,E1 -11028.594,E2 -11028.594} C_VEL
LIN {X 0,Y 403.147,Z 372.883,A -85,B 0,C 180,E1 -11030.089,E2 -11030.089} C_VEL
LIN {X 0,Y 403.425,Z 368.179,A -85,B 0,C 180,E1 -11031.622,E2 -11031.622} C_VEL
LIN {X 0,Y 403.822,Z 362.031,A -85,B 0,C 180,E1 -11033.184,E2 -11033.184} C_VEL
LIN {X 0,Y 404.384,Z 354.171,A -85,B 0,C 180,E1 -11034.769,E2 -11034.769} C_VEL
LIN {X 0,Y 405.048,Z 345.83,A -85,B 0,C 180,E1 -11036.124,E2 -11036.124} C_VEL
LIN {X 0,Y 405.741,Z 336.325,A -85,B 0,C 180,E1 -11037.376,E2 -11037.376} C_VEL
LIN {X 0,Y 406.433,Z 325.881,A -85,B 0,C 180,E1 -11038.491,E2 -11038.491} C_VEL
LIN {X 0,Y 407.155,Z 314.203,A -85,B 0,C 180,E1 -11039.485,E2 -11039.485} C_VEL
LIN {X 0,Y 407.851,Z 301.537,A -85,B 0,C 180,E1 -11040.304,E2 -11040.304} C_VEL
LIN {X 0,Y 408.342,Z 288.384,A -85,B 0,C 180,E1 -11040.926,E2 -11040.926} C_VEL
LIN {X 0,Y 408.716,Z 276.28,A -85,B 0,C 180,E1 -11041.306,E2 -11041.306} C_VEL
LIN {X 0,Y 409.943,Z 190.981,A -85,B 0,C 180,E1 -11042.911,E2 -11042.911} C_VEL
LIN {X 0,Y 405.982,Z 169.866,A -85,B 0,C 180,E1 -11043.527,E2 -11043.527} C_VEL
LIN {X 0,Y 406.168,Z 163.909,A -85,B 0,C 180,E1 -11044.918,E2 -11044.918} C_VEL
LIN {X 0,Y 404.18,Z 153.14,A -85,B 0,C 180,E1 -11047.644,E2 -11047.644} C_VEL
LIN {X 0,Y 404.155,Z 153.144,A -85,B 0,C 180,E1 -11050.708,E2 -11050.708} C_VEL
LIN {X 0,Y 404.17,Z 153.137,A -85,B 0,C 180,E1 -11053.012,E2 -11053.012} C_VEL
LIN {X 0,Y 403.51,Z 153.221,A -85,B 0,C 180,E1 -11053.844,E2 -11053.844} C_VEL
LIN {X 0,Y 400.683,Z 153.571,A -85,B 0,C 180,E1 -11055.196,E2 -11055.196} C_VEL
LIN {X 0,Y 398.295,Z 153.873,A -85,B 0,C 180,E1 -11056.289,E2 -11056.289} C_VEL
LIN {X 0,Y 397.279,Z 153.995,A -85,B 0,C 180,E1 -11057.133,E2 -11057.133} C_VEL
LIN {X 0,Y 397.201,Z 154.004,A -85,B 0,C 180,E1 -11057.419,E2 -11057.419} C_VEL
LIN {X 0,Y 397.223,Z 154.003,A -85,B 0,C 180,E1 -11060.838,E2 -11060.838} C_VEL
LIN {X 0,Y 397.323,Z 153.992,A -85,B 0,C 180,E1 -11063.908,E2 -11063.908} C_VEL
LIN {X 0,Y 397.436,Z 153.98,A -85,B 0,C 180,E1 -11067.973,E2 -11067.973} C_VEL
LIN {X 0,Y 397.434,Z 153.982,A -85,B 0,C 180,E1 -11072.027,E2 -11072.027} C_VEL
LIN {X 0,Y 397.316,Z 153.995,A -85,B 0,C 180,E1 -11076.092,E2 -11076.092} C_VEL
LIN {X 0,Y 397.223,Z 154.002,A -85,B 0,C 180,E1 -11079.163,E2 -11079.163} C_VEL
LIN {X 0,Y 397.21,Z 154.005,A -85,B 0,C 180,E1 -11082.258,E2 -11082.258} C_VEL
LIN {X 0,Y 397.119,Z 154.017,A -85,B 0,C 180,E1 -11085.394,E2 -11085.394} C_VEL
LIN {X 0,Y 397.083,Z 154.019,A -85,B 0,C 180,E1 -11088.577,E2 -11088.577} C_VEL
LIN {X 0,Y 397.086,Z 154.023,A -85,B 0,C 180,E1 -11091.819,E2 -11091.819} C_VEL
LIN {X 0,Y 397.098,Z 154.02,A -85,B 0,C 180,E1 -11095.135,E2 -11095.135} C_VEL
LIN {X 0,Y 397.056,Z 154.022,A -85,B 0,C 180,E1 -11098.549,E2 -11098.549} C_VEL
LIN {X 0,Y 397.072,Z 154.022,A -85,B 0,C 180,E1 -11101.835,E2 -11101.835} C_VEL
LIN {X 0,Y 397.115,Z 154.015,A -85,B 0,C 180,E1 -11104.494,E2 -11104.494} C_VEL
LIN {X 0,Y 397.086,Z 154.018,A -85,B 0,C 180,E1 -11108.276,E2 -11108.276} C_VEL
LIN {X 0,Y 397.046,Z 154.024,A -85,B 0,C 180,E1 -11111.976,E2 -11111.976} C_VEL
LIN {X 0,Y 397.081,Z 154.026,A -85,B 0,C 180,E1 -11115.069,E2 -11115.069} C_VEL
LIN {X 0,Y 397.046,Z 154.023,A -85,B 0,C 180,E1 -11118.024,E2 -11118.024} C_VEL
LIN {X 0,Y 397.084,Z 154.019,A -85,B 0,C 180,E1 -11121.723,E2 -11121.723} C_VEL
LIN {X 0,Y 397.11,Z 154.016,A -85,B 0,C 180,E1 -11125.506,E2 -11125.506} C_VEL
LIN {X 0,Y 397.07,Z 154.023,A -85,B 0,C 180,E1 -11129.117,E2 -11129.117} C_VEL
LIN {X 0,Y 397.055,Z 154.024,A -85,B 0,C 180,E1 -11132.252,E2 -11132.252} C_VEL
LIN {X 0,Y 397.097,Z 154.021,A -85,B 0,C 180,E1 -11134.865,E2 -11134.865} C_VEL
LIN {X 0,Y 397.086,Z 154.021,A -85,B 0,C 180,E1 -11138.181,E2 -11138.181} C_VEL
LIN {X 0,Y 397.108,Z 154.016,A -85,B 0,C 180,E1 -11141.424,E2 -11141.424} C_VEL
LIN {X 0,Y 397.118,Z 154.019,A -85,B 0,C 180,E1 -11144.606,E2 -11144.606} C_VEL
LIN {X 0,Y 397.208,Z 154.004,A -85,B 0,C 180,E1 -11147.742,E2 -11147.742} C_VEL
LIN {X 0,Y 397.22,Z 154.003,A -85,B 0,C 180,E1 -11150.838,E2 -11150.838} C_VEL
LIN {X 0,Y 397.313,Z 153.994,A -85,B 0,C 180,E1 -11153.908,E2 -11153.908} C_VEL
LIN {X 0,Y 397.432,Z 153.981,A -85,B 0,C 180,E1 -11157.974,E2 -11157.974} C_VEL
LIN {X 0,Y 397.312,Z 153.99,A -85,B 0,C 180,E1 -11161.014,E2 -11161.014} C_VEL
LIN {X 0,Y 397.291,Z 153.993,A -85,B 0,C 180,E1 -11163.043,E2 -11163.043} C_VEL
LIN {X 0,Y 397.314,Z 153.995,A -85,B 0,C 180,E1 -11166.093,E2 -11166.093} C_VEL
LIN {X 0,Y 397.222,Z 154.002,A -85,B 0,C 180,E1 -11169.163,E2 -11169.163} C_VEL
LIN {X 0,Y 397.209,Z 154.005,A -85,B 0,C 180,E1 -11172.259,E2 -11172.259} C_VEL
LIN {X 0,Y 397.118,Z 154.018,A -85,B 0,C 180,E1 -11175.395,E2 -11175.395} C_VEL
LIN {X 0,Y 397.083,Z 154.019,A -85,B 0,C 180,E1 -11178.578,E2 -11178.578} C_VEL
LIN {X 0,Y 397.086,Z 154.022,A -85,B 0,C 180,E1 -11181.82,E2 -11181.82} C_VEL
LIN {X 0,Y 397.099,Z 154.02,A -85,B 0,C 180,E1 -11185.136,E2 -11185.136} C_VEL
LIN {X 0,Y 397.057,Z 154.022,A -85,B 0,C 180,E1 -11188.549,E2 -11188.549} C_VEL
LIN {X 0,Y 397.074,Z 154.022,A -85,B 0,C 180,E1 -11191.836,E2 -11191.836} C_VEL
LIN {X 0,Y 397.114,Z 154.015,A -85,B 0,C 180,E1 -11194.495,E2 -11194.495} C_VEL
LIN {X 0,Y 397.087,Z 154.018,A -85,B 0,C 180,E1 -11198.277,E2 -11198.277} C_VEL
LIN {X 0,Y 397.049,Z 154.023,A -85,B 0,C 180,E1 -11201.977,E2 -11201.977} C_VEL
LIN {X 0,Y 397.084,Z 154.025,A -85,B 0,C 180,E1 -11205.07,E2 -11205.07} C_VEL
LIN {X 0,Y 397.05,Z 154.023,A -85,B 0,C 180,E1 -11208.024,E2 -11208.024} C_VEL
LIN {X 0,Y 397.089,Z 154.018,A -85,B 0,C 180,E1 -11211.724,E2 -11211.724} C_VEL
LIN {X 0,Y 397.116,Z 154.015,A -85,B 0,C 180,E1 -11215.506,E2 -11215.506} C_VEL
LIN {X 0,Y 397.073,Z 154.025,A -85,B 0,C 180,E1 -11219.117,E2 -11219.117} C_VEL
LIN {X 0,Y 397.116,Z 154.083,A -85,B 0,C 180,E1 -11222.126,E2 -11222.126} C_VEL
LIN {X 0,Y 399.602,Z 166.58,A -85,B 0,C 180,E1 -11225.033,E2 -11225.033} C_VEL
LIN {X 0,Y 400.212,Z 170.637,A -85,B 0,C 180,E1 -11225.946,E2 -11225.946} C_VEL
LIN {X 0,Y 398.983,Z 188.173,A -85,B 0,C 180,E1 -11229.642,E2 -11229.642} C_VEL
LIN {X 0,Y 398.751,Z 190.815,A -85,B 0,C 180,E1 -11230.192,E2 -11230.192} C_VEL
LIN {X 0,Y 402.934,Z 219.048,A -85,B 0,C 180,E1 -11230.948,E2 -11230.948} C_VEL
LIN {X 0,Y 401.727,Z 299.335,A -85,B 0,C 180,E1 -11232.501,E2 -11232.501} C_VEL
LIN {X 0,Y 401.211,Z 312.243,A -85,B 0,C 180,E1 -11232.938,E2 -11232.938} C_VEL
LIN {X 0,Y 400.594,Z 324.862,A -85,B 0,C 180,E1 -11233.567,E2 -11233.567} C_VEL
LIN {X 0,Y 399.858,Z 336.144,A -85,B 0,C 180,E1 -11234.322,E2 -11234.322} C_VEL
LIN {X 0,Y 398.994,Z 347.835,A -85,B 0,C 180,E1 -11235.333,E2 -11235.333} C_VEL
LIN {X 0,Y 398.267,Z 358.866,A -85,B 0,C 180,E1 -11236.537,E2 -11236.537} C_VEL
LIN {X 0,Y 397.611,Z 367.86,A -85,B 0,C 180,E1 -11237.754,E2 -11237.754} C_VEL
LIN {X 0,Y 396.846,Z 376.998,A -85,B 0,C 180,E1 -11239.283,E2 -11239.283} C_VEL
LIN {X 0,Y 396.385,Z 384.36,A -85,B 0,C 180,E1 -11240.818,E2 -11240.818} C_VEL
LIN {X 0,Y 396.064,Z 390.237,A -85,B 0,C 180,E1 -11242.352,E2 -11242.352} C_VEL
LIN {X 0,Y 395.825,Z 395.62,A -85,B 0,C 180,E1 -11244.199,E2 -11244.199} C_VEL
LIN {X 0,Y 395.774,Z 399.241,A -85,B 0,C 180,E1 -11245.927,E2 -11245.927} C_VEL
LIN {X 0,Y 395.729,Z 400.793,A -85,B 0,C 180,E1 -11246.946,E2 -11246.946} C_VEL
LIN {X 0,Y 395.764,Z 401.884,A -85,B 0,C 180,E1 -11247.965,E2 -11247.965} C_VEL
LIN {X 0,Y 395.792,Z 402.562,A -85,B 0,C 180,E1 -11248.982,E2 -11248.982} C_VEL
LIN {X 0,Y 395.78,Z 402.844,A -85,B 0,C 180,E1 -11250,E2 -11250} C_VEL
LIN {X 0,Y 395.792,Z 402.727,A -85,B 0,C 180,E1 -11251.017,E2 -11251.017} C_VEL
LIN {X 0,Y 395.762,Z 402.166,A -85,B 0,C 180,E1 -11252.035,E2 -11252.035} C_VEL
LIN {X 0,Y 395.774,Z 399.834,A -85,B 0,C 180,E1 -11254.073,E2 -11254.073} C_VEL
LIN {X 0,Y 395.825,Z 396.526,A -85,B 0,C 180,E1 -11255.8,E2 -11255.8} C_VEL
LIN {X 0,Y 396.079,Z 391.466,A -85,B 0,C 180,E1 -11257.647,E2 -11257.647} C_VEL
LIN {X 0,Y 396.504,Z 384.953,A -85,B 0,C 180,E1 -11259.436,E2 -11259.436} C_VEL
LIN {X 0,Y 397.065,Z 377.851,A -85,B 0,C 180,E1 -11260.968,E2 -11260.968} C_VEL
LIN {X 0,Y 397.931,Z 368.97,A -85,B 0,C 180,E1 -11262.494,E2 -11262.494} C_VEL
LIN {X 0,Y 398.668,Z 360.211,A -85,B 0,C 180,E1 -11263.725,E2 -11263.725} C_VEL
LIN {X 0,Y 399.434,Z 350.277,A -85,B 0,C 180,E1 -11264.872,E2 -11264.872} C_VEL
LIN {X 0,Y 400.386,Z 338.891,A -85,B 0,C 180,E1 -11265.918,E2 -11265.918} C_VEL
LIN {X 0,Y 401.298,Z 326.621,A -85,B 0,C 180,E1 -11266.796,E2 -11266.796} C_VEL
LIN {X 0,Y 402.101,Z 313.742,A -85,B 0,C 180,E1 -11267.482,E2 -11267.482} C_VEL
LIN {X 0,Y 402.735,Z 300.907,A -85,B 0,C 180,E1 -11267.945,E2 -11267.945} C_VEL
LIN {X 0,Y 403.223,Z 278.946,A -85,B 0,C 180,E1 -11268.41,E2 -11268.41} C_VEL
LIN {X 0,Y 404.158,Z 218.244,A -85,B 0,C 180,E1 -11269.6,E2 -11269.6} C_VEL
LIN {X 0,Y 400.907,Z 198.336,A -85,B 0,C 180,E1 -11270.203,E2 -11270.203} C_VEL
LIN {X 0,Y 399.249,Z 189.677,A -85,B 0,C 180,E1 -11270.497,E2 -11270.497} C_VEL
LIN {X 0,Y 400.471,Z 173.885,A -85,B 0,C 180,E1 -11273.805,E2 -11273.805} C_VEL
LIN {X 0,Y 400.564,Z 170.865,A -85,B 0,C 180,E1 -11274.455,E2 -11274.455} C_VEL
LIN {X 0,Y 398.393,Z 159.951,A -85,B 0,C 180,E1 -11277.016,E2 -11277.016} C_VEL
LIN {X 0,Y 397.112,Z 154.025,A -85,B 0,C 180,E1 -11278.493,E2 -11278.493} C_VEL
LIN {X 0,Y 397.072,Z 154.028,A -85,B 0,C 180,E1 -11282.071,E2 -11282.071} C_VEL
LIN {X 0,Y 397.096,Z 154.023,A -85,B 0,C 180,E1 -11285.498,E2 -11285.498} C_VEL
LIN {X 0,Y 397.089,Z 154.025,A -85,B 0,C 180,E1 -11288.853,E2 -11288.853} C_VEL
LIN {X 0,Y 397.052,Z 154.029,A -85,B 0,C 180,E1 -11292.268,E2 -11292.268} C_VEL
LIN {X 0,Y 397.081,Z 154.024,A -85,B 0,C 180,E1 -11295.069,E2 -11295.069} C_VEL
LIN {X 0,Y 397.047,Z 154.023,A -85,B 0,C 180,E1 -11298.023,E2 -11298.023} C_VEL
LIN {X 0,Y 397.085,Z 154.021,A -85,B 0,C 180,E1 -11301.723,E2 -11301.723} C_VEL
LIN {X 0,Y 397.112,Z 154.016,A -85,B 0,C 180,E1 -11305.505,E2 -11305.505} C_VEL
LIN {X 0,Y 397.067,Z 154.02,A -85,B 0,C 180,E1 -11309.116,E2 -11309.116} C_VEL
LIN {X 0,Y 397.054,Z 154.027,A -85,B 0,C 180,E1 -11312.252,E2 -11312.252} C_VEL
LIN {X 0,Y 397.097,Z 154.022,A -85,B 0,C 180,E1 -11314.864,E2 -11314.864} C_VEL
LIN {X 0,Y 397.084,Z 154.017,A -85,B 0,C 180,E1 -11318.18,E2 -11318.18} C_VEL
LIN {X 0,Y 397.081,Z 154.015,A -85,B 0,C 180,E1 -11321.422,E2 -11321.422} C_VEL
LIN {X 0,Y 397.116,Z 154.013,A -85,B 0,C 180,E1 -11324.605,E2 -11324.605} C_VEL
LIN {X 0,Y 397.207,Z 154.006,A -85,B 0,C 180,E1 -11327.741,E2 -11327.741} C_VEL
LIN {X 0,Y 397.22,Z 154.002,A -85,B 0,C 180,E1 -11330.837,E2 -11330.837} C_VEL
LIN {X 0,Y 397.312,Z 153.997,A -85,B 0,C 180,E1 -11333.907,E2 -11333.907} C_VEL
LIN {X 0,Y 397.431,Z 153.978,A -85,B 0,C 180,E1 -11337.973,E2 -11337.973} C_VEL
LIN {X 0,Y 397.431,Z 153.983,A -85,B 0,C 180,E1 -11342.026,E2 -11342.026} C_VEL
LIN {X 0,Y 397.287,Z 153.996,A -85,B 0,C 180,E1 -11346.463,E2 -11346.463} C_VEL
LIN {X 0,Y 397.219,Z 154.008,A -85,B 0,C 180,E1 -11349.162,E2 -11349.162} C_VEL
LIN {X 0,Y 397.206,Z 154.013,A -85,B 0,C 180,E1 -11352.258,E2 -11352.258} C_VEL
LIN {X 0,Y 397.115,Z 154.025,A -85,B 0,C 180,E1 -11355.394,E2 -11355.394} C_VEL
LIN {X 0,Y 397.104,Z 154.021,A -85,B 0,C 180,E1 -11358.576,E2 -11358.576} C_VEL
LIN {X 0,Y 397.126,Z 154.094,A -85,B 0,C 180,E1 -11359.513,E2 -11359.513} C_VEL
LIN {X 0,Y 399.413,Z 164.851,A -85,B 0,C 180,E1 -11362.229,E2 -11362.229} C_VEL
LIN {X 0,Y 399.857,Z 169.302,A -85,B 0,C 180,E1 -11363.295,E2 -11363.295} C_VEL
LIN {X 0,Y 399.784,Z 170.628,A -85,B 0,C 180,E1 -11363.594,E2 -11363.594} C_VEL
LIN {X 0,Y 404.5,Z 192.212,A -85,B 0,C 180,E1 -11364.336,E2 -11364.336} C_VEL
LIN {X 0,Y 402.999,Z 278.796,A -85,B 0,C 180,E1 -11366.056,E2 -11366.056} C_VEL
LIN {X 0,Y 402.452,Z 292.304,A -85,B 0,C 180,E1 -11366.53,E2 -11366.53} C_VEL
LIN {X 0,Y 401.896,Z 304.828,A -85,B 0,C 180,E1 -11367.184,E2 -11367.184} C_VEL
LIN {X 0,Y 401.141,Z 315.849,A -85,B 0,C 180,E1 -11367.947,E2 -11367.947} C_VEL
LIN {X 0,Y 400.285,Z 327.456,A -85,B 0,C 180,E1 -11368.979,E2 -11368.979} C_VEL
LIN {X 0,Y 399.411,Z 337.428,A -85,B 0,C 180,E1 -11370.082,E2 -11370.082} C_VEL
LIN {X 0,Y 398.603,Z 346.656,A -85,B 0,C 180,E1 -11371.341,E2 -11371.341} C_VEL
LIN {X 0,Y 397.865,Z 354.308,A -85,B 0,C 180,E1 -11372.611,E2 -11372.611} C_VEL
LIN {X 0,Y 397.222,Z 361.558,A -85,B 0,C 180,E1 -11374.087,E2 -11374.087} C_VEL
LIN {X 0,Y 396.665,Z 368.186,A -85,B 0,C 180,E1 -11375.78,E2 -11375.78} C_VEL
LIN {X 0,Y 396.177,Z 373.927,A -85,B 0,C 180,E1 -11377.735,E2 -11377.735} C_VEL
LIN {X 0,Y 395.844,Z 378.001,A -85,B 0,C 180,E1 -11379.729,E2 -11379.729} C_VEL
LIN {X 0,Y 395.635,Z 380.391,A -85,B 0,C 180,E1 -11381.749,E2 -11381.749} C_VEL
LIN {X 0,Y 395.586,Z 381.217,A -85,B 0,C 180,E1 -11383.858,E2 -11383.858} C_VEL
LIN {X 0,Y 395.598,Z 380.761,A -85,B 0,C 180,E1 -11385.285,E2 -11385.285} C_VEL
LIN {X 0,Y 395.683,Z 379.481,A -85,B 0,C 180,E1 -11386.737,E2 -11386.737} C_VEL
LIN {X 0,Y 395.79,Z 377.299,A -85,B 0,C 180,E1 -11388.226,E2 -11388.226} C_VEL
LIN {X 0,Y 396.01,Z 374.118,A -85,B 0,C 180,E1 -11389.739,E2 -11389.739} C_VEL
LIN {X 0,Y 396.254,Z 369.747,A -85,B 0,C 180,E1 -11391.295,E2 -11391.295} C_VEL
LIN {X 0,Y 396.709,Z 363.678,A -85,B 0,C 180,E1 -11392.963,E2 -11392.963} C_VEL
LIN {X 0,Y 397.187,Z 356.704,A -85,B 0,C 180,E1 -11394.482,E2 -11394.482} C_VEL
LIN {X 0,Y 397.82,Z 348.783,A -85,B 0,C 180,E1 -11395.871,E2 -11395.871} C_VEL
LIN {X 0,Y 398.482,Z 340.303,A -85,B 0,C 180,E1 -11397.093,E2 -11397.093} C_VEL
LIN {X 0,Y 399.17,Z 330.384,A -85,B 0,C 180,E1 -11398.265,E2 -11398.265} C_VEL
LIN {X 0,Y 399.893,Z 320.512,A -85,B 0,C 180,E1 -11399.213,E2 -11399.213} C_VEL
LIN {X 0,Y 400.537,Z 309.455,A -85,B 0,C 180,E1 -11400.068,E2 -11400.068} C_VEL
LIN {X 0,Y 401.166,Z 297.776,A -85,B 0,C 180,E1 -11400.76,E2 -11400.76} C_VEL
LIN {X 0,Y 401.592,Z 284.653,A -85,B 0,C 180,E1 -11401.321,E2 -11401.321} C_VEL
LIN {X 0,Y 401.988,Z 270.923,A -85,B 0,C 180,E1 -11401.683,E2 -11401.683} C_VEL
LIN {X 0,Y 403.157,Z 191.974,A -85,B 0,C 180,E1 -11403.189,E2 -11403.189} C_VEL
LIN {X 0,Y 399.046,Z 170.152,A -85,B 0,C 180,E1 -11403.814,E2 -11403.814} C_VEL
LIN {X 0,Y 399.185,Z 165.138,A -85,B 0,C 180,E1 -11405.005,E2 -11405.005} C_VEL
LIN {X 0,Y 397.122,Z 154.019,A -85,B 0,C 180,E1 -11407.842,E2 -11407.842} C_VEL
LIN {X 0,Y 397.11,Z 154.017,A -85,B 0,C 180,E1 -11411.424,E2 -11411.424} C_VEL
LIN {X 0,Y 397.12,Z 154.019,A -85,B 0,C 180,E1 -11414.606,E2 -11414.606} C_VEL
LIN {X 0,Y 397.201,Z 154.004,A -85,B 0,C 180,E1 -11417.419,E2 -11417.419} C_VEL
LIN {X 0,Y 396.541,Z 154.092,A -85,B 0,C 180,E1 -11418.265,E2 -11418.265} C_VEL
LIN {X 0,Y 393.684,Z 154.443,A -85,B 0,C 180,E1 -11419.64,E2 -11419.64} C_VEL
LIN {X 0,Y 391.287,Z 154.743,A -85,B 0,C 180,E1 -11420.752,E2 -11420.752} C_VEL
LIN {X 0,Y 390.295,Z 154.865,A -85,B 0,C 180,E1 -11421.611,E2 -11421.611} C_VEL
LIN {X 0,Y 390.235,Z 154.875,A -85,B 0,C 180,E1 -11421.902,E2 -11421.902} C_VEL
LIN {X 0,Y 390.198,Z 154.877,A -85,B 0,C 180,E1 -11424.833,E2 -11424.833} C_VEL
LIN {X 0,Y 390.403,Z 154.855,A -85,B 0,C 180,E1 -11427.937,E2 -11427.937} C_VEL
LIN {X 0,Y 390.4,Z 154.858,A -85,B 0,C 180,E1 -11432.063,E2 -11432.063} C_VEL
LIN {X 0,Y 390.271,Z 154.871,A -85,B 0,C 180,E1 -11436.203,E2 -11436.203} C_VEL
LIN {X 0,Y 390.182,Z 154.88,A -85,B 0,C 180,E1 -11439.329,E2 -11439.329} C_VEL
LIN {X 0,Y 390.192,Z 154.88,A -85,B 0,C 180,E1 -11443.438,E2 -11443.438} C_VEL
LIN {X 0,Y 390.068,Z 154.895,A -85,B 0,C 180,E1 -11447.271,E2 -11447.271} C_VEL
LIN {X 0,Y 390.065,Z 154.893,A -85,B 0,C 180,E1 -11450.462,E2 -11450.462} C_VEL
LIN {X 0,Y 390.053,Z 154.899,A -85,B 0,C 180,E1 -11453.353,E2 -11453.353} C_VEL
LIN {X 0,Y 390.025,Z 154.899,A -85,B 0,C 180,E1 -11456.775,E2 -11456.775} C_VEL
LIN {X 0,Y 390.029,Z 154.898,A -85,B 0,C 180,E1 -11460.3,E2 -11460.3} C_VEL
LIN {X 0,Y 390.064,Z 154.894,A -85,B 0,C 180,E1 -11464.025,E2 -11464.025} C_VEL
LIN {X 0,Y 390.034,Z 154.9,A -85,B 0,C 180,E1 -11467.55,E2 -11467.55} C_VEL
LIN {X 0,Y 390.011,Z 154.903,A -85,B 0,C 180,E1 -11470.814,E2 -11470.814} C_VEL
LIN {X 0,Y 390.039,Z 154.897,A -85,B 0,C 180,E1 -11473.884,E2 -11473.884} C_VEL
LIN {X 0,Y 390.041,Z 154.9,A -85,B 0,C 180,E1 -11476.788,E2 -11476.788} C_VEL
LIN {X 0,Y 390.004,Z 154.902,A -85,B 0,C 180,E1 -11479.555,E2 -11479.555} C_VEL
LIN {X 0,Y 390.032,Z 154.899,A -85,B 0,C 180,E1 -11482.451,E2 -11482.451} C_VEL
LIN {X 0,Y 390.056,Z 154.894,A -85,B 0,C 180,E1 -11486.045,E2 -11486.045} C_VEL
LIN {X 0,Y 390.037,Z 154.897,A -85,B 0,C 180,E1 -11489.87,E2 -11489.87} C_VEL
LIN {X 0,Y 390.024,Z 154.899,A -85,B 0,C 180,E1 -11493.226,E2 -11493.226} C_VEL
LIN {X 0,Y 390.053,Z 154.899,A -85,B 0,C 180,E1 -11496.767,E2 -11496.767} C_VEL
LIN {X 0,Y 390.079,Z 154.893,A -85,B 0,C 180,E1 -11499.982,E2 -11499.982} C_VEL
LIN {X 0,Y 390.101,Z 154.889,A -85,B 0,C 180,E1 -11503.247,E2 -11503.247} C_VEL
LIN {X 0,Y 390.19,Z 154.882,A -85,B 0,C 180,E1 -11506.562,E2 -11506.562} C_VEL
LIN {X 0,Y 390.179,Z 154.881,A -85,B 0,C 180,E1 -11510.671,E2 -11510.671} C_VEL
LIN {X 0,Y 390.269,Z 154.87,A -85,B 0,C 180,E1 -11513.798,E2 -11513.798} C_VEL
LIN {X 0,Y 390.398,Z 154.856,A -85,B 0,C 180,E1 -11517.937,E2 -11517.937} C_VEL
LIN {X 0,Y 390.398,Z 154.858,A -85,B 0,C 180,E1 -11522.064,E2 -11522.064} C_VEL
LIN {X 0,Y 390.269,Z 154.871,A -85,B 0,C 180,E1 -11526.203,E2 -11526.203} C_VEL
LIN {X 0,Y 390.18,Z 154.88,A -85,B 0,C 180,E1 -11529.33,E2 -11529.33} C_VEL
LIN {X 0,Y 390.191,Z 154.881,A -85,B 0,C 180,E1 -11533.439,E2 -11533.439} C_VEL
LIN {X 0,Y 390.067,Z 154.895,A -85,B 0,C 180,E1 -11537.271,E2 -11537.271} C_VEL
LIN {X 0,Y 390.045,Z 154.898,A -85,B 0,C 180,E1 -11541.123,E2 -11541.123} C_VEL
LIN {X 0,Y 390.038,Z 154.896,A -85,B 0,C 180,E1 -11544.484,E2 -11544.484} C_VEL
LIN {X 0,Y 390.012,Z 154.901,A -85,B 0,C 180,E1 -11547.998,E2 -11547.998} C_VEL
LIN {X 0,Y 390.016,Z 154.904,A -85,B 0,C 180,E1 -11551.506,E2 -11551.506} C_VEL
LIN {X 0,Y 390.066,Z 154.899,A -85,B 0,C 180,E1 -11555.209,E2 -11555.209} C_VEL
LIN {X 0,Y 390.055,Z 154.9,A -85,B 0,C 180,E1 -11559.097,E2 -11559.097} C_VEL
LIN {X 0,Y 390.028,Z 154.898,A -85,B 0,C 180,E1 -11562.372,E2 -11562.372} C_VEL
LIN {X 0,Y 390.04,Z 154.899,A -85,B 0,C 180,E1 -11565.354,E2 -11565.354} C_VEL
LIN {X 0,Y 390.013,Z 154.9,A -85,B 0,C 180,E1 -11568.185,E2 -11568.185} C_VEL
LIN {X 0,Y 390.056,Z 154.901,A -85,B 0,C 180,E1 -11570.904,E2 -11570.904} C_VEL
LIN {X 0,Y 390.068,Z 154.899,A -85,B 0,C 180,E1 -11574.792,E2 -11574.792} C_VEL
LIN {X 0,Y 390.018,Z 154.903,A -85,B 0,C 180,E1 -11578.496,E2 -11578.496} C_VEL
LIN {X 0,Y 390.031,Z 154.951,A -85,B 0,C 180,E1 -11581.866,E2 -11581.866} C_VEL
LIN {X 0,Y 392.326,Z 166.18,A -85,B 0,C 180,E1 -11584.537,E2 -11584.537} C_VEL
LIN {X 0,Y 393.249,Z 171.978,A -85,B 0,C 180,E1 -11585.872,E2 -11585.872} C_VEL
LIN {X 0,Y 391.875,Z 190.508,A -85,B 0,C 180,E1 -11589.842,E2 -11589.842} C_VEL
LIN {X 0,Y 392.415,Z 194.741,A -85,B 0,C 180,E1 -11589.988,E2 -11589.988} C_VEL
LIN {X 0,Y 396.145,Z 219.532,A -85,B 0,C 180,E1 -11590.665,E2 -11590.665} C_VEL
LIN {X 0,Y 394.889,Z 298.711,A -85,B 0,C 180,E1 -11592.222,E2 -11592.222} C_VEL
LIN {X 0,Y 394.365,Z 311.752,A -85,B 0,C 180,E1 -11592.666,E2 -11592.666} C_VEL
LIN {X 0,Y 393.688,Z 325.001,A -85,B 0,C 180,E1 -11593.337,E2 -11593.337} C_VEL
LIN {X 0,Y 392.862,Z 336.982,A -85,B 0,C 180,E1 -11594.168,E2 -11594.168} C_VEL
LIN {X 0,Y 391.978,Z 348.487,A -85,B 0,C 180,E1 -11595.197,E2 -11595.197} C_VEL
LIN {X 0,Y 391.304,Z 358.532,A -85,B 0,C 180,E1 -11596.321,E2 -11596.321} C_VEL
LIN {X 0,Y 390.634,Z 367.379,A -85,B 0,C 180,E1 -11597.532,E2 -11597.532} C_VEL
LIN {X 0,Y 389.834,Z 376.571,A -85,B 0,C 180,E1 -11599.088,E2 -11599.088} C_VEL
LIN {X 0,Y 389.348,Z 383.978,A -85,B 0,C 180,E1 -11600.65,E2 -11600.65} C_VEL
LIN {X 0,Y 388.998,Z 389.899,A -85,B 0,C 180,E1 -11602.212,E2 -11602.212} C_VEL
LIN {X 0,Y 388.793,Z 394.694,A -85,B 0,C 180,E1 -11603.833,E2 -11603.833} C_VEL
LIN {X 0,Y 388.737,Z 396.985,A -85,B 0,C 180,E1 -11604.814,E2 -11604.814} C_VEL
LIN {X 0,Y 388.699,Z 398.977,A -85,B 0,C 180,E1 -11605.852,E2 -11605.852} C_VEL
LIN {X 0,Y 388.637,Z 400.544,A -85,B 0,C 180,E1 -11606.89,E2 -11606.89} C_VEL
LIN {X 0,Y 388.663,Z 401.658,A -85,B 0,C 180,E1 -11607.927,E2 -11607.927} C_VEL
LIN {X 0,Y 388.704,Z 402.349,A -85,B 0,C 180,E1 -11608.964,E2 -11608.964} C_VEL
LIN {X 0,Y 388.71,Z 402.642,A -85,B 0,C 180,E1 -11610,E2 -11610} C_VEL
LIN {X 0,Y 388.704,Z 402.539,A -85,B 0,C 180,E1 -11611.036,E2 -11611.036} C_VEL
LIN {X 0,Y 388.66,Z 401.996,A -85,B 0,C 180,E1 -11612.072,E2 -11612.072} C_VEL
LIN {X 0,Y 388.699,Z 399.684,A -85,B 0,C 180,E1 -11614.147,E2 -11614.147} C_VEL
LIN {X 0,Y 388.726,Z 396.727,A -85,B 0,C 180,E1 -11615.749,E2 -11615.749} C_VEL
LIN {X 0,Y 388.939,Z 392.912,A -85,B 0,C 180,E1 -11617.266,E2 -11617.266} C_VEL
LIN {X 0,Y 389.266,Z 387.865,A -85,B 0,C 180,E1 -11618.827,E2 -11618.827} C_VEL
LIN {X 0,Y 389.79,Z 381.528,A -85,B 0,C 180,E1 -11620.387,E2 -11620.387} C_VEL
LIN {X 0,Y 390.464,Z 373.617,A -85,B 0,C 180,E1 -11621.946,E2 -11621.946} C_VEL
LIN {X 0,Y 391.502,Z 363.771,A -85,B 0,C 180,E1 -11623.495,E2 -11623.495} C_VEL
LIN {X 0,Y 392.282,Z 353.816,A -85,B 0,C 180,E1 -11624.764,E2 -11624.764} C_VEL
LIN {X 0,Y 393.2,Z 343.506,A -85,B 0,C 180,E1 -11625.817,E2 -11625.817} C_VEL
LIN {X 0,Y 394.279,Z 330.826,A -85,B 0,C 180,E1 -11626.837,E2 -11626.837} C_VEL
LIN {X 0,Y 395.193,Z 318.198,A -85,B 0,C 180,E1 -11627.597,E2 -11627.597} C_VEL
LIN {X 0,Y 395.908,Z 304.873,A -85,B 0,C 180,E1 -11628.165,E2 -11628.165} C_VEL
LIN {X 0,Y 396.386,Z 291.983,A -85,B 0,C 180,E1 -11628.51,E2 -11628.51} C_VEL
LIN {X 0,Y 397.63,Z 219.498,A -85,B 0,C 180,E1 -11629.951,E2 -11629.951} C_VEL
LIN {X 0,Y 394.417,Z 199.716,A -85,B 0,C 180,E1 -11630.569,E2 -11630.569} C_VEL
LIN {X 0,Y 392.431,Z 189.397,A -85,B 0,C 180,E1 -11630.942,E2 -11630.942} C_VEL
LIN {X 0,Y 393.706,Z 173.955,A -85,B 0,C 180,E1 -11634.24,E2 -11634.24} C_VEL
LIN {X 0,Y 392.857,Z 167.815,A -85,B 0,C 180,E1 -11635.666,E2 -11635.666} C_VEL
LIN {X 0,Y 390.062,Z 154.905,A -85,B 0,C 180,E1 -11638.869,E2 -11638.869} C_VEL
LIN {X 0,Y 390.038,Z 154.904,A -85,B 0,C 180,E1 -11642.721,E2 -11642.721} C_VEL
LIN {X 0,Y 390.04,Z 154.901,A -85,B 0,C 180,E1 -11645.821,E2 -11645.821} C_VEL
LIN {X 0,Y 390.034,Z 154.906,A -85,B 0,C 180,E1 -11649.211,E2 -11649.211} C_VEL
LIN {X 0,Y 390.027,Z 154.905,A -85,B 0,C 180,E1 -11652.371,E2 -11652.371} C_VEL
LIN {X 0,Y 390.037,Z 154.902,A -85,B 0,C 180,E1 -11655.353,E2 -11655.353} C_VEL
LIN {X 0,Y 390.011,Z 154.9,A -85,B 0,C 180,E1 -11658.183,E2 -11658.183} C_VEL
LIN {X 0,Y 390.053,Z 154.897,A -85,B 0,C 180,E1 -11660.903,E2 -11660.903} C_VEL
LIN {X 0,Y 390.064,Z 154.899,A -85,B 0,C 180,E1 -11664.79,E2 -11664.79} C_VEL
LIN {X 0,Y 390.014,Z 154.904,A -85,B 0,C 180,E1 -11668.494,E2 -11668.494} C_VEL
LIN {X 0,Y 390.01,Z 154.902,A -85,B 0,C 180,E1 -11672.002,E2 -11672.002} C_VEL
LIN {X 0,Y 390.036,Z 154.899,A -85,B 0,C 180,E1 -11675.516,E2 -11675.516} C_VEL
LIN {X 0,Y 390.043,Z 154.9,A -85,B 0,C 180,E1 -11678.877,E2 -11678.877} C_VEL
LIN {X 0,Y 390.065,Z 154.897,A -85,B 0,C 180,E1 -11682.729,E2 -11682.729} C_VEL
LIN {X 0,Y 390.189,Z 154.882,A -85,B 0,C 180,E1 -11686.561,E2 -11686.561} C_VEL
LIN {X 0,Y 390.178,Z 154.881,A -85,B 0,C 180,E1 -11690.67,E2 -11690.67} C_VEL
LIN {X 0,Y 390.267,Z 154.873,A -85,B 0,C 180,E1 -11693.797,E2 -11693.797} C_VEL
LIN {X 0,Y 390.399,Z 154.854,A -85,B 0,C 180,E1 -11697.936,E2 -11697.936} C_VEL
LIN {X 0,Y 390.399,Z 154.858,A -85,B 0,C 180,E1 -11702.063,E2 -11702.063} C_VEL
LIN {X 0,Y 390.248,Z 154.874,A -85,B 0,C 180,E1 -11706.454,E2 -11706.454} C_VEL
LIN {X 0,Y 390.177,Z 154.886,A -85,B 0,C 180,E1 -11709.329,E2 -11709.329} C_VEL
LIN {X 0,Y 390.188,Z 154.889,A -85,B 0,C 180,E1 -11713.438,E2 -11713.438} C_VEL
LIN {X 0,Y 390.098,Z 154.897,A -85,B 0,C 180,E1 -11717.287,E2 -11717.287} C_VEL
LIN {X 0,Y 390.102,Z 154.968,A -85,B 0,C 180,E1 -11719.126,E2 -11719.126} C_VEL
LIN {X 0,Y 392.513,Z 166.426,A -85,B 0,C 180,E1 -11722.086,E2 -11722.086} C_VEL
LIN {X 0,Y 392.998,Z 170.862,A -85,B 0,C 180,E1 -11723.167,E2 -11723.167} C_VEL
LIN {X 0,Y 397.819,Z 192.558,A -85,B 0,C 180,E1 -11723.947,E2 -11723.947} C_VEL
LIN {X 0,Y 398.019,Z 195.912,A -85,B 0,C 180,E1 -11724.03,E2 -11724.03} C_VEL
LIN {X 0,Y 396.337,Z 279.265,A -85,B 0,C 180,E1 -11725.711,E2 -11725.711} C_VEL
LIN {X 0,Y 395.794,Z 292.583,A -85,B 0,C 180,E1 -11726.19,E2 -11726.19} C_VEL
LIN {X 0,Y 395.181,Z 305.425,A -85,B 0,C 180,E1 -11726.876,E2 -11726.876} C_VEL
LIN {X 0,Y 394.295,Z 317.598,A -85,B 0,C 180,E1 -11727.752,E2 -11727.752} C_VEL
LIN {X 0,Y 393.297,Z 329.399,A -85,B 0,C 180,E1 -11728.847,E2 -11728.847} C_VEL
LIN {X 0,Y 392.365,Z 339.982,A -85,B 0,C 180,E1 -11730.101,E2 -11730.101} C_VEL
LIN {X 0,Y 391.533,Z 348.687,A -85,B 0,C 180,E1 -11731.368,E2 -11731.368} C_VEL
LIN {X 0,Y 390.6,Z 357.63,A -85,B 0,C 180,E1 -11732.975,E2 -11732.975} C_VEL
LIN {X 0,Y 389.935,Z 364.765,A -85,B 0,C 180,E1 -11734.604,E2 -11734.604} C_VEL
LIN {X 0,Y 389.48,Z 370.029,A -85,B 0,C 180,E1 -11736.107,E2 -11736.107} C_VEL
LIN {X 0,Y 389.064,Z 374.855,A -85,B 0,C 180,E1 -11737.891,E2 -11737.891} C_VEL
LIN {X 0,Y 388.839,Z 377.558,A -85,B 0,C 180,E1 -11739.242,E2 -11739.242} C_VEL
LIN {X 0,Y 388.679,Z 379.566,A -85,B 0,C 180,E1 -11740.612,E2 -11740.612} C_VEL
LIN {X 0,Y 388.533,Z 380.932,A -85,B 0,C 180,E1 -11742.131,E2 -11742.131} C_VEL
LIN {X 0,Y 388.486,Z 381.403,A -85,B 0,C 180,E1 -11743.646,E2 -11743.646} C_VEL
LIN {X 0,Y 388.508,Z 381.025,A -85,B 0,C 180,E1 -11745.131,E2 -11745.131} C_VEL
LIN {X 0,Y 388.59,Z 379.855,A -85,B 0,C 180,E1 -11746.587,E2 -11746.587} C_VEL
LIN {X 0,Y 388.686,Z 377.936,A -85,B 0,C 180,E1 -11748.01,E2 -11748.01} C_VEL
LIN {X 0,Y 388.862,Z 375.236,A -85,B 0,C 180,E1 -11749.411,E2 -11749.411} C_VEL
LIN {X 0,Y 389.117,Z 371.27,A -85,B 0,C 180,E1 -11750.953,E2 -11750.953} C_VEL
LIN {X 0,Y 389.509,Z 365.958,A -85,B 0,C 180,E1 -11752.551,E2 -11752.551} C_VEL
LIN {X 0,Y 389.983,Z 359.016,A -85,B 0,C 180,E1 -11754.189,E2 -11754.189} C_VEL
LIN {X 0,Y 390.688,Z 350.211,A -85,B 0,C 180,E1 -11755.84,E2 -11755.84} C_VEL
LIN {X 0,Y 391.492,Z 340.652,A -85,B 0,C 180,E1 -11757.263,E2 -11757.263} C_VEL
LIN {X 0,Y 392.287,Z 329.907,A -85,B 0,C 180,E1 -11758.548,E2 -11758.548} C_VEL
LIN {X 0,Y 393.055,Z 319.362,A -85,B 0,C 180,E1 -11759.559,E2 -11759.559} C_VEL
LIN {X 0,Y 393.796,Z 307.074,A -85,B 0,C 180,E1 -11760.479,E2 -11760.479} C_VEL
LIN {X 0,Y 394.417,Z 294.908,A -85,B 0,C 180,E1 -11761.165,E2 -11761.165} C_VEL
LIN {X 0,Y 394.864,Z 282.087,A -85,B 0,C 180,E1 -11761.678,E2 -11761.678} C_VEL
LIN {X 0,Y 395.18,Z 265.452,A -85,B 0,C 180,E1 -11762.063,E2 -11762.063} C_VEL
LIN {X 0,Y 396.387,Z 192.905,A -85,B 0,C 180,E1 -11763.472,E2 -11763.472} C_VEL
LIN {X 0,Y 392.145,Z 170.219,A -85,B 0,C 180,E1 -11764.164,E2 -11764.164} C_VEL
LIN {X 0,Y 392.224,Z 166.349,A -85,B 0,C 180,E1 -11765.098,E2 -11765.098} C_VEL
LIN {X 0,Y 390.093,Z 154.895,A -85,B 0,C 180,E1 -11768.083,E2 -11768.083} C_VEL
LIN {X 0,Y 390.066,Z 154.897,A -85,B 0,C 180,E1 -11771.076,E2 -11771.076} C_VEL
LIN {X 0,Y 390.063,Z 154.899,A -85,B 0,C 180,E1 -11774.32,E2 -11774.32} C_VEL
LIN {X 0,Y 390.163,Z 154.881,A -85,B 0,C 180,E1 -11777.517,E2 -11777.517} C_VEL
LIN {X 0,Y 390.182,Z 154.881,A -85,B 0,C 180,E1 -11780.671,E2 -11780.671} C_VEL
LIN {X 0,Y 390.235,Z 154.875,A -85,B 0,C 180,E1 -11781.902,E2 -11781.902} C_VEL
LIN {X 0,Y 389.589,Z 154.96,A -85,B 0,C 180,E1 -11782.764,E2 -11782.764} C_VEL
LIN {X 0,Y 386.631,Z 155.328,A -85,B 0,C 180,E1 -11784.162,E2 -11784.162} C_VEL
LIN {X 0,Y 384.151,Z 155.632,A -85,B 0,C 180,E1 -11785.293,E2 -11785.293} C_VEL
LIN {X 0,Y 383.158,Z 155.76,A -85,B 0,C 180,E1 -11786.17,E2 -11786.17} C_VEL
LIN {X 0,Y 383.118,Z 155.758,A -85,B 0,C 180,E1 -11786.467,E2 -11786.467} C_VEL
LIN {X 0,Y 383.369,Z 155.731,A -85,B 0,C 180,E1 -11787.899,E2 -11787.899} C_VEL
LIN {X 0,Y 383.365,Z 155.734,A -85,B 0,C 180,E1 -11792.101,E2 -11792.101} C_VEL
LIN {X 0,Y 383.229,Z 155.747,A -85,B 0,C 180,E1 -11796.317,E2 -11796.317} C_VEL
LIN {X 0,Y 383.133,Z 155.759,A -85,B 0,C 180,E1 -11799.503,E2 -11799.503} C_VEL
LIN {X 0,Y 383.123,Z 155.762,A -85,B 0,C 180,E1 -11803.536,E2 -11803.536} C_VEL
LIN {X 0,Y 383.02,Z 155.774,A -85,B 0,C 180,E1 -11807.42,E2 -11807.42} C_VEL
LIN {X 0,Y 383.009,Z 155.772,A -85,B 0,C 180,E1 -11810.64,E2 -11810.64} C_VEL
LIN {X 0,Y 383.003,Z 155.777,A -85,B 0,C 180,E1 -11813.809,E2 -11813.809} C_VEL
LIN {X 0,Y 382.963,Z 155.783,A -85,B 0,C 180,E1 -11817.309,E2 -11817.309} C_VEL
LIN {X 0,Y 382.974,Z 155.778,A -85,B 0,C 180,E1 -11820.919,E2 -11820.919} C_VEL
LIN {X 0,Y 383.012,Z 155.773,A -85,B 0,C 180,E1 -11824.668,E2 -11824.668} C_VEL
LIN {X 0,Y 382.988,Z 155.775,A -85,B 0,C 180,E1 -11827.902,E2 -11827.902} C_VEL
LIN {X 0,Y 382.955,Z 155.783,A -85,B 0,C 180,E1 -11831.351,E2 -11831.351} C_VEL
LIN {X 0,Y 382.984,Z 155.775,A -85,B 0,C 180,E1 -11834.302,E2 -11834.302} C_VEL
LIN {X 0,Y 382.991,Z 155.779,A -85,B 0,C 180,E1 -11837.238,E2 -11837.238} C_VEL
LIN {X 0,Y 382.98,Z 155.777,A -85,B 0,C 180,E1 -11840.419,E2 -11840.419} C_VEL
LIN {X 0,Y 383.007,Z 155.772,A -85,B 0,C 180,E1 -11844.043,E2 -11844.043} C_VEL
LIN {X 0,Y 382.979,Z 155.776,A -85,B 0,C 180,E1 -11847.579,E2 -11847.579} C_VEL
LIN {X 0,Y 382.969,Z 155.779,A -85,B 0,C 180,E1 -11850.299,E2 -11850.299} C_VEL
LIN {X 0,Y 382.997,Z 155.775,A -85,B 0,C 180,E1 -11854.045,E2 -11854.045} C_VEL
LIN {X 0,Y 382.979,Z 155.776,A -85,B 0,C 180,E1 -11857.334,E2 -11857.334} C_VEL
LIN {X 0,Y 383.028,Z 155.774,A -85,B 0,C 180,E1 -11860.715,E2 -11860.715} C_VEL
LIN {X 0,Y 383.014,Z 155.774,A -85,B 0,C 180,E1 -11864.024,E2 -11864.024} C_VEL
LIN {X 0,Y 383.128,Z 155.757,A -85,B 0,C 180,E1 -11867.284,E2 -11867.284} C_VEL
LIN {X 0,Y 383.13,Z 155.761,A -85,B 0,C 180,E1 -11870.498,E2 -11870.498} C_VEL
LIN {X 0,Y 383.227,Z 155.746,A -85,B 0,C 180,E1 -11873.683,E2 -11873.683} C_VEL
LIN {X 0,Y 383.363,Z 155.732,A -85,B 0,C 180,E1 -11877.899,E2 -11877.899} C_VEL
LIN {X 0,Y 383.363,Z 155.734,A -85,B 0,C 180,E1 -11882.102,E2 -11882.102} C_VEL
LIN {X 0,Y 383.227,Z 155.747,A -85,B 0,C 180,E1 -11886.318,E2 -11886.318} C_VEL
LIN {X 0,Y 383.132,Z 155.76,A -85,B 0,C 180,E1 -11889.503,E2 -11889.503} C_VEL
LIN {X 0,Y 383.122,Z 155.762,A -85,B 0,C 180,E1 -11893.536,E2 -11893.536} C_VEL
LIN {X 0,Y 383.02,Z 155.775,A -85,B 0,C 180,E1 -11897.421,E2 -11897.421} C_VEL
LIN {X 0,Y 383.01,Z 155.772,A -85,B 0,C 180,E1 -11900.641,E2 -11900.641} C_VEL
LIN {X 0,Y 383.004,Z 155.776,A -85,B 0,C 180,E1 -11903.81,E2 -11903.81} C_VEL
LIN {X 0,Y 382.964,Z 155.783,A -85,B 0,C 180,E1 -11907.309,E2 -11907.309} C_VEL
LIN {X 0,Y 382.976,Z 155.778,A -85,B 0,C 180,E1 -11910.92,E2 -11910.92} C_VEL
LIN {X 0,Y 383.009,Z 155.773,A -85,B 0,C 180,E1 -11914.669,E2 -11914.669} C_VEL
LIN {X 0,Y 382.99,Z 155.775,A -85,B 0,C 180,E1 -11917.903,E2 -11917.903} C_VEL
LIN {X 0,Y 382.958,Z 155.783,A -85,B 0,C 180,E1 -11921.351,E2 -11921.351} C_VEL
LIN {X 0,Y 382.988,Z 155.775,A -85,B 0,C 180,E1 -11924.303,E2 -11924.303} C_VEL
LIN {X 0,Y 382.981,Z 155.78,A -85,B 0,C 180,E1 -11927.237,E2 -11927.237} C_VEL
LIN {X 0,Y 382.985,Z 155.777,A -85,B 0,C 180,E1 -11930.42,E2 -11930.42} C_VEL
LIN {X 0,Y 383.013,Z 155.772,A -85,B 0,C 180,E1 -11934.044,E2 -11934.044} C_VEL
LIN {X 0,Y 382.983,Z 155.777,A -85,B 0,C 180,E1 -11937.58,E2 -11937.58} C_VEL
LIN {X 0,Y 382.976,Z 155.779,A -85,B 0,C 180,E1 -11940.299,E2 -11940.299} C_VEL
LIN {X 0,Y 383.015,Z 155.937,A -85,B 0,C 180,E1 -11941.634,E2 -11941.634} C_VEL
LIN {X 0,Y 385.509,Z 168.337,A -85,B 0,C 180,E1 -11944.633,E2 -11944.633} C_VEL
LIN {X 0,Y 386.189,Z 171.991,A -85,B 0,C 180,E1 -11945.495,E2 -11945.495} C_VEL
LIN {X 0,Y 385.734,Z 179.821,A -85,B 0,C 180,E1 -11947.222,E2 -11947.222} C_VEL
LIN {X 0,Y 384.94,Z 190.422,A -85,B 0,C 180,E1 -11949.529,E2 -11949.529} C_VEL
LIN {X 0,Y 389.366,Z 220.713,A -85,B 0,C 180,E1 -11950.386,E2 -11950.386} C_VEL
LIN {X 0,Y 388.03,Z 299.199,A -85,B 0,C 180,E1 -11951.965,E2 -11951.965} C_VEL
LIN {X 0,Y 387.45,Z 312.759,A -85,B 0,C 180,E1 -11952.449,E2 -11952.449} C_VEL
LIN {X 0,Y 386.784,Z 325.128,A -85,B 0,C 180,E1 -11953.099,E2 -11953.099} C_VEL
LIN {X 0,Y 385.868,Z 337.817,A -85,B 0,C 180,E1 -11954.009,E2 -11954.009} C_VEL
LIN {X 0,Y 384.962,Z 349.138,A -85,B 0,C 180,E1 -11955.056,E2 -11955.056} C_VEL
LIN {X 0,Y 384.259,Z 359.352,A -85,B 0,C 180,E1 -11956.245,E2 -11956.245} C_VEL
LIN {X 0,Y 383.511,Z 368.554,A -85,B 0,C 180,E1 -11957.566,E2 -11957.566} C_VEL
LIN {X 0,Y 382.71,Z 377.519,A -85,B 0,C 180,E1 -11959.151,E2 -11959.151} C_VEL
LIN {X 0,Y 382.217,Z 384.696,A -85,B 0,C 180,E1 -11960.741,E2 -11960.741} C_VEL
LIN {X 0,Y 381.858,Z 391.228,A -85,B 0,C 180,E1 -11962.598,E2 -11962.598} C_VEL
LIN {X 0,Y 381.693,Z 394.775,A -85,B 0,C 180,E1 -11963.876,E2 -11963.876} C_VEL
LIN {X 0,Y 381.624,Z 398.712,A -85,B 0,C 180,E1 -11965.775,E2 -11965.775} C_VEL
LIN {X 0,Y 381.548,Z 400.293,A -85,B 0,C 180,E1 -11966.832,E2 -11966.832} C_VEL
LIN {X 0,Y 381.562,Z 401.432,A -85,B 0,C 180,E1 -11967.889,E2 -11967.889} C_VEL
LIN {X 0,Y 381.618,Z 402.135,A -85,B 0,C 180,E1 -11968.945,E2 -11968.945} C_VEL
LIN {X 0,Y 381.641,Z 402.441,A -85,B 0,C 180,E1 -11970,E2 -11970} C_VEL
LIN {X 0,Y 381.603,Z 402.349,A -85,B 0,C 180,E1 -11971.055,E2 -11971.055} C_VEL
LIN {X 0,Y 381.558,Z 401.827,A -85,B 0,C 180,E1 -11972.111,E2 -11972.111} C_VEL
LIN {X 0,Y 381.624,Z 399.533,A -85,B 0,C 180,E1 -11974.224,E2 -11974.224} C_VEL
LIN {X 0,Y 381.67,Z 396.105,A -85,B 0,C 180,E1 -11976.092,E2 -11976.092} C_VEL
LIN {X 0,Y 381.977,Z 391.269,A -85,B 0,C 180,E1 -11977.931,E2 -11977.931} C_VEL
LIN {X 0,Y 382.467,Z 384.811,A -85,B 0,C 180,E1 -11979.786,E2 -11979.786} C_VEL
LIN {X 0,Y 383.059,Z 377.79,A -85,B 0,C 180,E1 -11981.375,E2 -11981.375} C_VEL
LIN {X 0,Y 384.029,Z 369.007,A -85,B 0,C 180,E1 -11982.955,E2 -11982.955} C_VEL
LIN {X 0,Y 384.85,Z 359.949,A -85,B 0,C 180,E1 -11984.283,E2 -11984.283} C_VEL
LIN {X 0,Y 385.872,Z 348.979,A -85,B 0,C 180,E1 -11985.583,E2 -11985.583} C_VEL
LIN {X 0,Y 386.949,Z 337.825,A -85,B 0,C 180,E1 -11986.622,E2 -11986.622} C_VEL
LIN {X 0,Y 387.962,Z 325.39,A -85,B 0,C 180,E1 -11987.527,E2 -11987.527} C_VEL
LIN {X 0,Y 388.796,Z 312.851,A -85,B 0,C 180,E1 -11988.202,E2 -11988.202} C_VEL
LIN {X 0,Y 389.516,Z 298.746,A -85,B 0,C 180,E1 -11988.712,E2 -11988.712} C_VEL
LIN {X 0,Y 390.977,Z 219.752,A -85,B 0,C 180,E1 -11990.349,E2 -11990.349} C_VEL
LIN {X 0,Y 387.663,Z 199.342,A -85,B 0,C 180,E1 -11991.011,E2 -11991.011} C_VEL
LIN {X 0,Y 385.647,Z 189.257,A -85,B 0,C 180,E1 -11991.375,E2 -11991.375} C_VEL
LIN {X 0,Y 386.849,Z 174.863,A -85,B 0,C 180,E1 -11994.512,E2 -11994.512} C_VEL
LIN {X 0,Y 385.454,Z 166.93,A -85,B 0,C 180,E1 -11996.435,E2 -11996.435} C_VEL
LIN {X 0,Y 382.991,Z 155.789,A -85,B 0,C 180,E1 -11999.284,E2 -11999.284} C_VEL
LIN {X 0,Y 382.982,Z 155.784,A -85,B 0,C 180,E1 -12002.42,E2 -12002.42} C_VEL
LIN {X 0,Y 383.011,Z 155.776,A -85,B 0,C 180,E1 -12005.956,E2 -12005.956} C_VEL
LIN {X 0,Y 382.983,Z 155.783,A -85,B 0,C 180,E1 -12009.58,E2 -12009.58} C_VEL
LIN {X 0,Y 383.004,Z 155.779,A -85,B 0,C 180,E1 -12012.778,E2 -12012.778} C_VEL
LIN {X 0,Y 382.986,Z 155.779,A -85,B 0,C 180,E1 -12015.787,E2 -12015.787} C_VEL
LIN {X 0,Y 382.958,Z 155.784,A -85,B 0,C 180,E1 -12018.8,E2 -12018.8} C_VEL
LIN {X 0,Y 382.988,Z 155.778,A -85,B 0,C 180,E1 -12022.097,E2 -12022.097} C_VEL
LIN {X 0,Y 383.007,Z 155.774,A -85,B 0,C 180,E1 -12025.33,E2 -12025.33} C_VEL
LIN {X 0,Y 382.974,Z 155.776,A -85,B 0,C 180,E1 -12029.08,E2 -12029.08} C_VEL
LIN {X 0,Y 382.962,Z 155.778,A -85,B 0,C 180,E1 -12032.69,E2 -12032.69} C_VEL
LIN {X 0,Y 383.002,Z 155.778,A -85,B 0,C 180,E1 -12036.19,E2 -12036.19} C_VEL
LIN {X 0,Y 383.03,Z 155.772,A -85,B 0,C 180,E1 -12039.597,E2 -12039.597} C_VEL
LIN {X 0,Y 383.034,Z 155.772,A -85,B 0,C 180,E1 -12042.928,E2 -12042.928} C_VEL
LIN {X 0,Y 383.12,Z 155.764,A -85,B 0,C 180,E1 -12046.463,E2 -12046.463} C_VEL
LIN {X 0,Y 383.129,Z 155.76,A -85,B 0,C 180,E1 -12050.497,E2 -12050.497} C_VEL
LIN {X 0,Y 383.225,Z 155.75,A -85,B 0,C 180,E1 -12053.682,E2 -12053.682} C_VEL
LIN {X 0,Y 383.365,Z 155.73,A -85,B 0,C 180,E1 -12057.898,E2 -12057.898} C_VEL
LIN {X 0,Y 383.364,Z 155.734,A -85,B 0,C 180,E1 -12062.101,E2 -12062.101} C_VEL
LIN {X 0,Y 383.214,Z 155.751,A -85,B 0,C 180,E1 -12066.442,E2 -12066.442} C_VEL
LIN {X 0,Y 383.128,Z 155.764,A -85,B 0,C 180,E1 -12069.502,E2 -12069.502} C_VEL
LIN {X 0,Y 383.118,Z 155.771,A -85,B 0,C 180,E1 -12073.536,E2 -12073.536} C_VEL
LIN {X 0,Y 383.063,Z 155.772,A -85,B 0,C 180,E1 -12077.442,E2 -12077.442} C_VEL
LIN {X 0,Y 383.054,Z 155.863,A -85,B 0,C 180,E1 -12078.728,E2 -12078.728} C_VEL
LIN {X 0,Y 385.38,Z 166.536,A -85,B 0,C 180,E1 -12081.558,E2 -12081.558} C_VEL
LIN {X 0,Y 386.154,Z 171.155,A -85,B 0,C 180,E1 -12082.717,E2 -12082.717} C_VEL
LIN {X 0,Y 390.097,Z 187.771,A -85,B 0,C 180,E1 -12083.35,E2 -12083.35} C_VEL
LIN {X 0,Y 391.515,Z 194.868,A -85,B 0,C 180,E1 -12083.598,E2 -12083.598} C_VEL
LIN {X 0,Y 389.707,Z 279.295,A -85,B 0,C 180,E1 -12085.342,E2 -12085.342} C_VEL
LIN {X 0,Y 389.129,Z 292.716,A -85,B 0,C 180,E1 -12085.83,E2 -12085.83} C_VEL
LIN {X 0,Y 388.491,Z 305.548,A -85,B 0,C 180,E1 -12086.526,E2 -12086.526} C_VEL
LIN {X 0,Y 387.535,Z 318.083,A -85,B 0,C 180,E1 -12087.445,E2 -12087.445} C_VEL
LIN {X 0,Y 386.579,Z 329.187,A -85,B 0,C 180,E1 -12088.491,E2 -12088.491} C_VEL
LIN {X 0,Y 385.644,Z 338.835,A -85,B 0,C 180,E1 -12089.625,E2 -12089.625} C_VEL
LIN {X 0,Y 384.67,Z 348.766,A -85,B 0,C 180,E1 -12091.077,E2 -12091.077} C_VEL
LIN {X 0,Y 383.739,Z 357.194,A -85,B 0,C 180,E1 -12092.6,E2 -12092.6} C_VEL
LIN {X 0,Y 383.175,Z 362.811,A -85,B 0,C 180,E1 -12093.846,E2 -12093.846} C_VEL
LIN {X 0,Y 382.544,Z 369.506,A -85,B 0,C 180,E1 -12095.683,E2 -12095.683} C_VEL
LIN {X 0,Y 382.098,Z 374.191,A -85,B 0,C 180,E1 -12097.371,E2 -12097.371} C_VEL
LIN {X 0,Y 381.743,Z 378.162,A -85,B 0,C 180,E1 -12099.356,E2 -12099.356} C_VEL
LIN {X 0,Y 381.542,Z 380.233,A -85,B 0,C 180,E1 -12100.957,E2 -12100.957} C_VEL
LIN {X 0,Y 381.373,Z 381.52,A -85,B 0,C 180,E1 -12102.987,E2 -12102.987} C_VEL
LIN {X 0,Y 381.402,Z 381.498,A -85,B 0,C 180,E1 -12104.444,E2 -12104.444} C_VEL
LIN {X 0,Y 381.442,Z 380.67,A -85,B 0,C 180,E1 -12105.936,E2 -12105.936} C_VEL
LIN {X 0,Y 381.555,Z 378.994,A -85,B 0,C 180,E1 -12107.457,E2 -12107.457} C_VEL
LIN {X 0,Y 381.692,Z 376.358,A -85,B 0,C 180,E1 -12109.018,E2 -12109.018} C_VEL
LIN {X 0,Y 381.978,Z 372.661,A -85,B 0,C 180,E1 -12110.601,E2 -12110.601} C_VEL
LIN {X 0,Y 382.367,Z 367.715,A -85,B 0,C 180,E1 -12112.217,E2 -12112.217} C_VEL
LIN {X 0,Y 382.837,Z 360.629,A -85,B 0,C 180,E1 -12114.025,E2 -12114.025} C_VEL
LIN {X 0,Y 383.48,Z 352.988,A -85,B 0,C 180,E1 -12115.558,E2 -12115.558} C_VEL
LIN {X 0,Y 384.251,Z 343.982,A -85,B 0,C 180,E1 -12117.017,E2 -12117.017} C_VEL
LIN {X 0,Y 385.128,Z 333.314,A -85,B 0,C 180,E1 -12118.41,E2 -12118.41} C_VEL
LIN {X 0,Y 385.926,Z 322.853,A -85,B 0,C 180,E1 -12119.495,E2 -12119.495} C_VEL
LIN {X 0,Y 386.678,Z 311.153,A -85,B 0,C 180,E1 -12120.462,E2 -12120.462} C_VEL
LIN {X 0,Y 387.363,Z 299.747,A -85,B 0,C 180,E1 -12121.189,E2 -12121.189} C_VEL
LIN {X 0,Y 387.87,Z 286.977,A -85,B 0,C 180,E1 -12121.784,E2 -12121.784} C_VEL
LIN {X 0,Y 388.26,Z 273.483,A -85,B 0,C 180,E1 -12122.185,E2 -12122.185} C_VEL
LIN {X 0,Y 389.547,Z 193.578,A -85,B 0,C 180,E1 -12123.774,E2 -12123.774} C_VEL
LIN {X 0,Y 385.25,Z 170.487,A -85,B 0,C 180,E1 -12124.471,E2 -12124.471} C_VEL
LIN {X 0,Y 385.249,Z 167.565,A -85,B 0,C 180,E1 -12125.192,E2 -12125.192} C_VEL
LIN {X 0,Y 383.015,Z 155.777,A -85,B 0,C 180,E1 -12128.33,E2 -12128.33} C_VEL
LIN {X 0,Y 383.016,Z 155.772,A -85,B 0,C 180,E1 -12131.825,E2 -12131.825} C_VEL
LIN {X 0,Y 383.024,Z 155.771,A -85,B 0,C 180,E1 -12135.115,E2 -12135.115} C_VEL
LIN {X 0,Y 383.13,Z 155.757,A -85,B 0,C 180,E1 -12137.284,E2 -12137.284} C_VEL
LIN {X 0,Y 383.132,Z 155.761,A -85,B 0,C 180,E1 -12140.498,E2 -12140.498} C_VEL
LIN {X 0,Y 383.235,Z 155.745,A -85,B 0,C 180,E1 -12143.683,E2 -12143.683} C_VEL
LIN {X 0,Y 383.118,Z 155.758,A -85,B 0,C 180,E1 -12146.467,E2 -12146.467} C_VEL
LIN {X 0,Y 382.563,Z 155.829,A -85,B 0,C 180,E1 -12147.345,E2 -12147.345} C_VEL
LIN {X 0,Y 379.758,Z 156.179,A -85,B 0,C 180,E1 -12148.773,E2 -12148.773} C_VEL
LIN {X 0,Y 377.33,Z 156.484,A -85,B 0,C 180,E1 -12149.927,E2 -12149.927} C_VEL
LIN {X 0,Y 376.301,Z 156.608,A -85,B 0,C 180,E1 -12150.821,E2 -12150.821} C_VEL
LIN {X 0,Y 376.229,Z 156.616,A -85,B 0,C 180,E1 -12151.123,E2 -12151.123} C_VEL
LIN {X 0,Y 376.329,Z 156.61,A -85,B 0,C 180,E1 -12152.141,E2 -12152.141} C_VEL
LIN {X 0,Y 376.189,Z 156.623,A -85,B 0,C 180,E1 -12156.436,E2 -12156.436} C_VEL
LIN {X 0,Y 376.104,Z 156.637,A -85,B 0,C 180,E1 -12159.682,E2 -12159.682} C_VEL
LIN {X 0,Y 376.087,Z 156.64,A -85,B 0,C 180,E1 -12163.657,E2 -12163.657} C_VEL
LIN {X 0,Y 375.979,Z 156.653,A -85,B 0,C 180,E1 -12167.577,E2 -12167.577} C_VEL
LIN {X 0,Y 375.975,Z 156.649,A -85,B 0,C 180,E1 -12170.832,E2 -12170.832} C_VEL
LIN {X 0,Y 375.93,Z 156.654,A -85,B 0,C 180,E1 -12174.286,E2 -12174.286} C_VEL
LIN {X 0,Y 375.906,Z 156.657,A -85,B 0,C 180,E1 -12176.661,E2 -12176.661} C_VEL
LIN {X 0,Y 375.908,Z 156.659,A -85,B 0,C 180,E1 -12179.084,E2 -12179.084} C_VEL
LIN {X 0,Y 375.95,Z 156.656,A -85,B 0,C 180,E1 -12181.562,E2 -12181.562} C_VEL
LIN {X 0,Y 375.951,Z 156.657,A -85,B 0,C 180,E1 -12185.416,E2 -12185.416} C_VEL
LIN {X 0,Y 375.93,Z 156.654,A -85,B 0,C 180,E1 -12188.263,E2 -12188.263} C_VEL
LIN {X 0,Y 375.908,Z 156.659,A -85,B 0,C 180,E1 -12191.597,E2 -12191.597} C_VEL
LIN {X 0,Y 375.916,Z 156.659,A -85,B 0,C 180,E1 -12194.73,E2 -12194.73} C_VEL
LIN {X 0,Y 375.911,Z 156.657,A -85,B 0,C 180,E1 -12197.698,E2 -12197.698} C_VEL
LIN {X 0,Y 375.928,Z 156.656,A -85,B 0,C 180,E1 -12200.534,E2 -12200.534} C_VEL
LIN {X 0,Y 375.951,Z 156.652,A -85,B 0,C 180,E1 -12203.497,E2 -12203.497} C_VEL
LIN {X 0,Y 375.952,Z 156.651,A -85,B 0,C 180,E1 -12205.888,E2 -12205.888} C_VEL
LIN {X 0,Y 375.955,Z 156.651,A -85,B 0,C 180,E1 -12209.687,E2 -12209.687} C_VEL
LIN {X 0,Y 375.911,Z 156.658,A -85,B 0,C 180,E1 -12212.135,E2 -12212.135} C_VEL
LIN {X 0,Y 375.93,Z 156.659,A -85,B 0,C 180,E1 -12214.534,E2 -12214.534} C_VEL
LIN {X 0,Y 375.964,Z 156.653,A -85,B 0,C 180,E1 -12216.887,E2 -12216.887} C_VEL
LIN {X 0,Y 375.969,Z 156.654,A -85,B 0,C 180,E1 -12220.338,E2 -12220.338} C_VEL
LIN {X 0,Y 375.969,Z 156.65,A -85,B 0,C 180,E1 -12223.717,E2 -12223.717} C_VEL
LIN {X 0,Y 376.097,Z 156.634,A -85,B 0,C 180,E1 -12227.042,E2 -12227.042} C_VEL
LIN {X 0,Y 376.101,Z 156.639,A -85,B 0,C 180,E1 -12230.319,E2 -12230.319} C_VEL
LIN {X 0,Y 376.187,Z 156.623,A -85,B 0,C 180,E1 -12233.564,E2 -12233.564} C_VEL
LIN {X 0,Y 376.327,Z 156.608,A -85,B 0,C 180,E1 -12237.86,E2 -12237.86} C_VEL
LIN {X 0,Y 376.327,Z 156.61,A -85,B 0,C 180,E1 -12242.141,E2 -12242.141} C_VEL
LIN {X 0,Y 376.187,Z 156.623,A -85,B 0,C 180,E1 -12246.436,E2 -12246.436} C_VEL
LIN {X 0,Y 376.102,Z 156.637,A -85,B 0,C 180,E1 -12249.682,E2 -12249.682} C_VEL
LIN {X 0,Y 376.086,Z 156.64,A -85,B 0,C 180,E1 -12253.658,E2 -12253.658} C_VEL
LIN {X 0,Y 375.978,Z 156.654,A -85,B 0,C 180,E1 -12257.577,E2 -12257.577} C_VEL
LIN {X 0,Y 375.976,Z 156.649,A -85,B 0,C 180,E1 -12260.833,E2 -12260.833} C_VEL
LIN {X 0,Y 375.931,Z 156.654,A -85,B 0,C 180,E1 -12264.286,E2 -12264.286} C_VEL
LIN {X 0,Y 375.907,Z 156.657,A -85,B 0,C 180,E1 -12266.661,E2 -12266.661} C_VEL
LIN {X 0,Y 375.909,Z 156.66,A -85,B 0,C 180,E1 -12269.085,E2 -12269.085} C_VEL
LIN {X 0,Y 375.951,Z 156.655,A -85,B 0,C 180,E1 -12271.563,E2 -12271.563} C_VEL
LIN {X 0,Y 375.946,Z 156.657,A -85,B 0,C 180,E1 -12275.417,E2 -12275.417} C_VEL
LIN {X 0,Y 375.932,Z 156.654,A -85,B 0,C 180,E1 -12278.263,E2 -12278.263} C_VEL
LIN {X 0,Y 375.912,Z 156.658,A -85,B 0,C 180,E1 -12281.597,E2 -12281.597} C_VEL
LIN {X 0,Y 375.919,Z 156.658,A -85,B 0,C 180,E1 -12284.731,E2 -12284.731} C_VEL
LIN {X 0,Y 375.906,Z 156.657,A -85,B 0,C 180,E1 -12287.697,E2 -12287.697} C_VEL
LIN {X 0,Y 375.934,Z 156.656,A -85,B 0,C 180,E1 -12290.534,E2 -12290.534} C_VEL
LIN {X 0,Y 375.957,Z 156.651,A -85,B 0,C 180,E1 -12293.498,E2 -12293.498} C_VEL
LIN {X 0,Y 375.957,Z 156.65,A -85,B 0,C 180,E1 -12295.889,E2 -12295.889} C_VEL
LIN {X 0,Y 375.96,Z 156.652,A -85,B 0,C 180,E1 -12299.687,E2 -12299.687} C_VEL
LIN {X 0,Y 375.95,Z 156.677,A -85,B 0,C 180,E1 -12301.334,E2 -12301.334} C_VEL
LIN {X 0,Y 378.472,Z 169.195,A -85,B 0,C 180,E1 -12304.422,E2 -12304.422} C_VEL
LIN {X 0,Y 379.274,Z 174.187,A -85,B 0,C 180,E1 -12305.615,E2 -12305.615} C_VEL
LIN {X 0,Y 378.029,Z 190.276,A -85,B 0,C 180,E1 -12309.194,E2 -12309.194} C_VEL
LIN {X 0,Y 382.602,Z 221.47,A -85,B 0,C 180,E1 -12310.089,E2 -12310.089} C_VEL
LIN {X 0,Y 381.229,Z 298.509,A -85,B 0,C 180,E1 -12311.666,E2 -12311.666} C_VEL
LIN {X 0,Y 380.645,Z 312.221,A -85,B 0,C 180,E1 -12312.159,E2 -12312.159} C_VEL
LIN {X 0,Y 379.966,Z 324.124,A -85,B 0,C 180,E1 -12312.786,E2 -12312.786} C_VEL
LIN {X 0,Y 379.156,Z 335.456,A -85,B 0,C 180,E1 -12313.58,E2 -12313.58} C_VEL
LIN {X 0,Y 378.185,Z 347.176,A -85,B 0,C 180,E1 -12314.644,E2 -12314.644} C_VEL
LIN {X 0,Y 377.441,Z 357.326,A -85,B 0,C 180,E1 -12315.801,E2 -12315.801} C_VEL
LIN {X 0,Y 376.661,Z 366.382,A -85,B 0,C 180,E1 -12317.062,E2 -12317.062} C_VEL
LIN {X 0,Y 375.942,Z 374.331,A -85,B 0,C 180,E1 -12318.407,E2 -12318.407} C_VEL
LIN {X 0,Y 375.327,Z 382.075,A -85,B 0,C 180,E1 -12320.026,E2 -12320.026} C_VEL
LIN {X 0,Y 375,Z 387.371,A -85,B 0,C 180,E1 -12321.377,E2 -12321.377} C_VEL
LIN {X 0,Y 374.725,Z 392.482,A -85,B 0,C 180,E1 -12322.998,E2 -12322.998} C_VEL
LIN {X 0,Y 374.55,Z 396.424,A -85,B 0,C 180,E1 -12324.617,E2 -12324.617} C_VEL
LIN {X 0,Y 374.551,Z 398.448,A -85,B 0,C 180,E1 -12325.695,E2 -12325.695} C_VEL
LIN {X 0,Y 374.462,Z 400.042,A -85,B 0,C 180,E1 -12326.772,E2 -12326.772} C_VEL
LIN {X 0,Y 374.461,Z 401.205,A -85,B 0,C 180,E1 -12327.849,E2 -12327.849} C_VEL
LIN {X 0,Y 374.519,Z 401.921,A -85,B 0,C 180,E1 -12328.925,E2 -12328.925} C_VEL
LIN {X 0,Y 374.556,Z 402.238,A -85,B 0,C 180,E1 -12330,E2 -12330} C_VEL
LIN {X 0,Y 374.504,Z 402.157,A -85,B 0,C 180,E1 -12331.075,E2 -12331.075} C_VEL
LIN {X 0,Y 374.457,Z 401.659,A -85,B 0,C 180,E1 -12332.151,E2 -12332.151} C_VEL
LIN {X 0,Y 374.46,Z 400.725,A -85,B 0,C 180,E1 -12333.228,E2 -12333.228} C_VEL
LIN {X 0,Y 374.528,Z 399.391,A -85,B 0,C 180,E1 -12334.304,E2 -12334.304} C_VEL
LIN {X 0,Y 374.566,Z 396.335,A -85,B 0,C 180,E1 -12336.041,E2 -12336.041} C_VEL
LIN {X 0,Y 374.822,Z 392.721,A -85,B 0,C 180,E1 -12337.542,E2 -12337.542} C_VEL
LIN {X 0,Y 375.194,Z 387.733,A -85,B 0,C 180,E1 -12339.161,E2 -12339.161} C_VEL
LIN {X 0,Y 375.79,Z 381.463,A -85,B 0,C 180,E1 -12340.779,E2 -12340.779} C_VEL
LIN {X 0,Y 376.58,Z 373.668,A -85,B 0,C 180,E1 -12342.393,E2 -12342.393} C_VEL
LIN {X 0,Y 377.648,Z 363.901,A -85,B 0,C 180,E1 -12344,E2 -12344} C_VEL
LIN {X 0,Y 378.562,Z 353.846,A -85,B 0,C 180,E1 -12345.34,E2 -12345.34} C_VEL
LIN {X 0,Y 379.573,Z 343.933,A -85,B 0,C 180,E1 -12346.401,E2 -12346.401} C_VEL
LIN {X 0,Y 380.747,Z 331.484,A -85,B 0,C 180,E1 -12347.454,E2 -12347.454} C_VEL
LIN {X 0,Y 381.734,Z 319.346,A -85,B 0,C 180,E1 -12348.239,E2 -12348.239} C_VEL
LIN {X 0,Y 382.518,Z 306.766,A -85,B 0,C 180,E1 -12348.824,E2 -12348.824} C_VEL
LIN {X 0,Y 383.072,Z 293.987,A -85,B 0,C 180,E1 -12349.213,E2 -12349.213} C_VEL
LIN {X 0,Y 384.447,Z 220.44,A -85,B 0,C 180,E1 -12350.752,E2 -12350.752} C_VEL
LIN {X 0,Y 380.603,Z 197.434,A -85,B 0,C 180,E1 -12351.528,E2 -12351.528} C_VEL
LIN {X 0,Y 378.884,Z 188.943,A -85,B 0,C 180,E1 -12351.867,E2 -12351.867} C_VEL
LIN {X 0,Y 379.939,Z 177.113,A -85,B 0,C 180,E1 -12354.5,E2 -12354.5} C_VEL
LIN {X 0,Y 379.48,Z 172.931,A -85,B 0,C 180,E1 -12355.505,E2 -12355.505} C_VEL
LIN {X 0,Y 377.206,Z 162.051,A -85,B 0,C 180,E1 -12358.274,E2 -12358.274} C_VEL
LIN {X 0,Y 375.935,Z 156.667,A -85,B 0,C 180,E1 -12359.735,E2 -12359.735} C_VEL
LIN {X 0,Y 375.947,Z 156.659,A -85,B 0,C 180,E1 -12362.828,E2 -12362.828} C_VEL
LIN {X 0,Y 375.947,Z 156.657,A -85,B 0,C 180,E1 -12365.416,E2 -12365.416} C_VEL
LIN {X 0,Y 375.932,Z 156.659,A -85,B 0,C 180,E1 -12368.262,E2 -12368.262} C_VEL
LIN {X 0,Y 375.911,Z 156.664,A -85,B 0,C 180,E1 -12371.596,E2 -12371.596} C_VEL
LIN {X 0,Y 375.917,Z 156.661,A -85,B 0,C 180,E1 -12374.729,E2 -12374.729} C_VEL
LIN {X 0,Y 375.904,Z 156.657,A -85,B 0,C 180,E1 -12377.695,E2 -12377.695} C_VEL
LIN {X 0,Y 375.93,Z 156.654,A -85,B 0,C 180,E1 -12380.533,E2 -12380.533} C_VEL
LIN {X 0,Y 375.953,Z 156.649,A -85,B 0,C 180,E1 -12383.496,E2 -12383.496} C_VEL
LIN {X 0,Y 375.953,Z 156.652,A -85,B 0,C 180,E1 -12385.887,E2 -12385.887} C_VEL
LIN {X 0,Y 375.955,Z 156.648,A -85,B 0,C 180,E1 -12389.686,E2 -12389.686} C_VEL
LIN {X 0,Y 375.912,Z 156.659,A -85,B 0,C 180,E1 -12392.134,E2 -12392.134} C_VEL
LIN {X 0,Y 375.93,Z 156.654,A -85,B 0,C 180,E1 -12394.533,E2 -12394.533} C_VEL
LIN {X 0,Y 375.964,Z 156.646,A -85,B 0,C 180,E1 -12396.886,E2 -12396.886} C_VEL
LIN {X 0,Y 375.954,Z 156.651,A -85,B 0,C 180,E1 -12400.336,E2 -12400.336} C_VEL
LIN {X 0,Y 375.954,Z 156.654,A -85,B 0,C 180,E1 -12403.715,E2 -12403.715} C_VEL
LIN {X 0,Y 376.096,Z 156.635,A -85,B 0,C 180,E1 -12407.041,E2 -12407.041} C_VEL
LIN {X 0,Y 376.1,Z 156.638,A -85,B 0,C 180,E1 -12410.318,E2 -12410.318} C_VEL
LIN {X 0,Y 376.185,Z 156.626,A -85,B 0,C 180,E1 -12413.564,E2 -12413.564} C_VEL
LIN {X 0,Y 376.329,Z 156.606,A -85,B 0,C 180,E1 -12417.859,E2 -12417.859} C_VEL
LIN {X 0,Y 376.329,Z 156.61,A -85,B 0,C 180,E1 -12422.14,E2 -12422.14} C_VEL
LIN {X 0,Y 376.185,Z 156.626,A -85,B 0,C 180,E1 -12426.436,E2 -12426.436} C_VEL
LIN {X 0,Y 376.099,Z 156.639,A -85,B 0,C 180,E1 -12429.681,E2 -12429.681} C_VEL
LIN {X 0,Y 376.082,Z 156.648,A -85,B 0,C 180,E1 -12433.657,E2 -12433.657} C_VEL
LIN {X 0,Y 375.997,Z 156.652,A -85,B 0,C 180,E1 -12437.933,E2 -12437.933} C_VEL
LIN {X 0,Y 376.003,Z 156.78,A -85,B 0,C 180,E1 -12438.304,E2 -12438.304} C_VEL
LIN {X 0,Y 378.178,Z 166.518,A -85,B 0,C 180,E1 -12440.961,E2 -12440.961} C_VEL
LIN {X 0,Y 379.169,Z 171.584,A -85,B 0,C 180,E1 -12442.233,E2 -12442.233} C_VEL
LIN {X 0,Y 381.761,Z 180.435,A -85,B 0,C 180,E1 -12442.625,E2 -12442.625} C_VEL
LIN {X 0,Y 384.955,Z 195.469,A -85,B 0,C 180,E1 -12443.182,E2 -12443.182} C_VEL
LIN {X 0,Y 383.129,Z 279.466,A -85,B 0,C 180,E1 -12444.954,E2 -12444.954} C_VEL
LIN {X 0,Y 382.485,Z 293.3,A -85,B 0,C 180,E1 -12445.469,E2 -12445.469} C_VEL
LIN {X 0,Y 381.824,Z 305.489,A -85,B 0,C 180,E1 -12446.142,E2 -12446.142} C_VEL
LIN {X 0,Y 380.895,Z 317.412,A -85,B 0,C 180,E1 -12447.023,E2 -12447.023} C_VEL
LIN {X 0,Y 379.825,Z 329.278,A -85,B 0,C 180,E1 -12448.152,E2 -12448.152} C_VEL
LIN {X 0,Y 378.757,Z 339.782,A -85,B 0,C 180,E1 -12449.421,E2 -12449.421} C_VEL
LIN {X 0,Y 377.802,Z 348.805,A -85,B 0,C 180,E1 -12450.767,E2 -12450.767} C_VEL
LIN {X 0,Y 376.758,Z 357.824,A -85,B 0,C 180,E1 -12452.431,E2 -12452.431} C_VEL
LIN {X 0,Y 375.991,Z 364.962,A -85,B 0,C 180,E1 -12454.108,E2 -12454.108} C_VEL
LIN {X 0,Y 375.399,Z 370.997,A -85,B 0,C 180,E1 -12455.912,E2 -12455.912} C_VEL
LIN {X 0,Y 375,Z 374.959,A -85,B 0,C 180,E1 -12457.445,E2 -12457.445} C_VEL
LIN {X 0,Y 374.726,Z 377.871,A -85,B 0,C 180,E1 -12458.924,E2 -12458.924} C_VEL
LIN {X 0,Y 374.454,Z 380.651,A -85,B 0,C 180,E1 -12461.063,E2 -12461.063} C_VEL
LIN {X 0,Y 374.279,Z 381.718,A -85,B 0,C 180,E1 -12462.92,E2 -12462.92} C_VEL
LIN {X 0,Y 374.304,Z 381.682,A -85,B 0,C 180,E1 -12464.481,E2 -12464.481} C_VEL
LIN {X 0,Y 374.346,Z 380.808,A -85,B 0,C 180,E1 -12466.003,E2 -12466.003} C_VEL
LIN {X 0,Y 374.46,Z 379.163,A -85,B 0,C 180,E1 -12467.496,E2 -12467.496} C_VEL
LIN {X 0,Y 374.602,Z 376.774,A -85,B 0,C 180,E1 -12468.957,E2 -12468.957} C_VEL
LIN {X 0,Y 374.856,Z 373.597,A -85,B 0,C 180,E1 -12470.399,E2 -12470.399} C_VEL
LIN {X 0,Y 375.276,Z 368.254,A -85,B 0,C 180,E1 -12472.224,E2 -12472.224} C_VEL
LIN {X 0,Y 375.766,Z 361.211,A -85,B 0,C 180,E1 -12474.072,E2 -12474.072} C_VEL
LIN {X 0,Y 376.417,Z 353.829,A -85,B 0,C 180,E1 -12475.608,E2 -12475.608} C_VEL
LIN {X 0,Y 377.2,Z 345.11,A -85,B 0,C 180,E1 -12477.07,E2 -12477.07} C_VEL
LIN {X 0,Y 378.076,Z 334.71,A -85,B 0,C 180,E1 -12478.48,E2 -12478.48} C_VEL
LIN {X 0,Y 378.932,Z 323.99,A -85,B 0,C 180,E1 -12479.643,E2 -12479.643} C_VEL
LIN {X 0,Y 379.798,Z 311.475,A -85,B 0,C 180,E1 -12480.704,E2 -12480.704} C_VEL
LIN {X 0,Y 380.539,Z 299.375,A -85,B 0,C 180,E1 -12481.486,E2 -12481.486} C_VEL
LIN {X 0,Y 381.063,Z 285.959,A -85,B 0,C 180,E1 -12482.104,E2 -12482.104} C_VEL
LIN {X 0,Y 381.483,Z 272.125,A -85,B 0,C 180,E1 -12482.503,E2 -12482.503} C_VEL
LIN {X 0,Y 382.843,Z 194.721,A -85,B 0,C 180,E1 -12484.068,E2 -12484.068} C_VEL
LIN {X 0,Y 378.367,Z 170.583,A -85,B 0,C 180,E1 -12484.831,E2 -12484.831} C_VEL
LIN {X 0,Y 377.497,Z 164.54,A -85,B 0,C 180,E1 -12486.405,E2 -12486.405} C_VEL
LIN {X 0,Y 375.985,Z 156.652,A -85,B 0,C 180,E1 -12488.563,E2 -12488.563} C_VEL
LIN {X 0,Y 376.003,Z 156.651,A -85,B 0,C 180,E1 -12492.411,E2 -12492.411} C_VEL
LIN {X 0,Y 376.086,Z 156.641,A -85,B 0,C 180,E1 -12496.343,E2 -12496.343} C_VEL
LIN {X 0,Y 376.103,Z 156.639,A -85,B 0,C 180,E1 -12500.318,E2 -12500.318} C_VEL
LIN {X 0,Y 376.193,Z 156.622,A -85,B 0,C 180,E1 -12503.564,E2 -12503.564} C_VEL
LIN {X 0,Y 376.334,Z 156.607,A -85,B 0,C 180,E1 -12507.86,E2 -12507.86} C_VEL
LIN {X 0,Y 376.229,Z 156.616,A -85,B 0,C 180,E1 -12511.123,E2 -12511.123} C_VEL
LIN {X 0,Y 375.581,Z 156.704,A -85,B 0,C 180,E1 -12512.015,E2 -12512.015} C_VEL
LIN {X 0,Y 372.69,Z 157.059,A -85,B 0,C 180,E1 -12513.463,E2 -12513.463} C_VEL
LIN {X 0,Y 370.232,Z 157.365,A -85,B 0,C 180,E1 -12514.635,E2 -12514.635} C_VEL
LIN {X 0,Y 369.188,Z 157.496,A -85,B 0,C 180,E1 -12515.542,E2 -12515.542} C_VEL
LIN {X 0,Y 369.109,Z 157.503,A -85,B 0,C 180,E1 -12515.849,E2 -12515.849} C_VEL
LIN {X 0,Y 369.086,Z 157.507,A -85,B 0,C 180,E1 -12518.762,E2 -12518.762} C_VEL
LIN {X 0,Y 368.995,Z 157.521,A -85,B 0,C 180,E1 -12522.094,E2 -12522.094} C_VEL
LIN {X 0,Y 368.987,Z 157.52,A -85,B 0,C 180,E1 -12524.336,E2 -12524.336} C_VEL
LIN {X 0,Y 368.95,Z 157.529,A -85,B 0,C 180,E1 -12527.745,E2 -12527.745} C_VEL
LIN {X 0,Y 368.905,Z 157.531,A -85,B 0,C 180,E1 -12531.221,E2 -12531.221} C_VEL
LIN {X 0,Y 368.904,Z 157.532,A -85,B 0,C 180,E1 -12533.874,E2 -12533.874} C_VEL
LIN {X 0,Y 368.853,Z 157.539,A -85,B 0,C 180,E1 -12537.212,E2 -12537.212} C_VEL
LIN {X 0,Y 368.887,Z 157.535,A -85,B 0,C 180,E1 -12539.692,E2 -12539.692} C_VEL
LIN {X 0,Y 368.891,Z 157.534,A -85,B 0,C 180,E1 -12543.043,E2 -12543.043} C_VEL
LIN {X 0,Y 368.911,Z 157.528,A -85,B 0,C 180,E1 -12546.197,E2 -12546.197} C_VEL
LIN {X 0,Y 368.869,Z 157.537,A -85,B 0,C 180,E1 -12548.957,E2 -12548.957} C_VEL
LIN {X 0,Y 368.853,Z 157.536,A -85,B 0,C 180,E1 -12552.005,E2 -12552.005} C_VEL
LIN {X 0,Y 368.869,Z 157.539,A -85,B 0,C 180,E1 -12555.175,E2 -12555.175} C_VEL
LIN {X 0,Y 368.859,Z 157.535,A -85,B 0,C 180,E1 -12558.175,E2 -12558.175} C_VEL
LIN {X 0,Y 368.87,Z 157.536,A -85,B 0,C 180,E1 -12561.366,E2 -12561.366} C_VEL
LIN {X 0,Y 368.925,Z 157.53,A -85,B 0,C 180,E1 -12565.146,E2 -12565.146} C_VEL
LIN {X 0,Y 368.908,Z 157.532,A -85,B 0,C 180,E1 -12569.045,E2 -12569.045} C_VEL
LIN {X 0,Y 368.901,Z 157.53,A -85,B 0,C 180,E1 -12571.558,E2 -12571.558} C_VEL
LIN {X 0,Y 368.88,Z 157.533,A -85,B 0,C 180,E1 -12575.22,E2 -12575.22} C_VEL
LIN {X 0,Y 368.89,Z 157.531,A -85,B 0,C 180,E1 -12577.603,E2 -12577.603} C_VEL
LIN {X 0,Y 368.91,Z 157.529,A -85,B 0,C 180,E1 -12581.104,E2 -12581.104} C_VEL
LIN {X 0,Y 368.934,Z 157.531,A -85,B 0,C 180,E1 -12584.533,E2 -12584.533} C_VEL
LIN {X 0,Y 369.052,Z 157.513,A -85,B 0,C 180,E1 -12586.79,E2 -12586.79} C_VEL
LIN {X 0,Y 369.052,Z 157.516,A -85,B 0,C 180,E1 -12590.132,E2 -12590.132} C_VEL
LIN {X 0,Y 369.149,Z 157.499,A -85,B 0,C 180,E1 -12593.441,E2 -12593.441} C_VEL
LIN {X 0,Y 369.29,Z 157.484,A -85,B 0,C 180,E1 -12597.819,E2 -12597.819} C_VEL
LIN {X 0,Y 369.197,Z 157.493,A -85,B 0,C 180,E1 -12601.091,E2 -12601.091} C_VEL
LIN {X 0,Y 369.29,Z 157.486,A -85,B 0,C 180,E1 -12602.182,E2 -12602.182} C_VEL
LIN {X 0,Y 369.149,Z 157.499,A -85,B 0,C 180,E1 -12606.56,E2 -12606.56} C_VEL
LIN {X 0,Y 369.053,Z 157.517,A -85,B 0,C 180,E1 -12609.869,E2 -12609.869} C_VEL
LIN {X 0,Y 369.034,Z 157.519,A -85,B 0,C 180,E1 -12613.772,E2 -12613.772} C_VEL
LIN {X 0,Y 368.95,Z 157.529,A -85,B 0,C 180,E1 -12617.745,E2 -12617.745} C_VEL
LIN {X 0,Y 368.905,Z 157.532,A -85,B 0,C 180,E1 -12621.222,E2 -12621.222} C_VEL
LIN {X 0,Y 368.904,Z 157.532,A -85,B 0,C 180,E1 -12623.874,E2 -12623.874} C_VEL
LIN {X 0,Y 368.854,Z 157.539,A -85,B 0,C 180,E1 -12627.213,E2 -12627.213} C_VEL
LIN {X 0,Y 368.889,Z 157.534,A -85,B 0,C 180,E1 -12629.693,E2 -12629.693} C_VEL
LIN {X 0,Y 368.893,Z 157.534,A -85,B 0,C 180,E1 -12633.043,E2 -12633.043} C_VEL
LIN {X 0,Y 368.909,Z 157.529,A -85,B 0,C 180,E1 -12636.198,E2 -12636.198} C_VEL
LIN {X 0,Y 368.871,Z 157.537,A -85,B 0,C 180,E1 -12638.958,E2 -12638.958} C_VEL
LIN {X 0,Y 368.857,Z 157.535,A -85,B 0,C 180,E1 -12642.006,E2 -12642.006} C_VEL
LIN {X 0,Y 368.873,Z 157.538,A -85,B 0,C 180,E1 -12645.175,E2 -12645.175} C_VEL
LIN {X 0,Y 368.859,Z 157.535,A -85,B 0,C 180,E1 -12648.175,E2 -12648.175} C_VEL
LIN {X 0,Y 368.875,Z 157.535,A -85,B 0,C 180,E1 -12651.367,E2 -12651.367} C_VEL
LIN {X 0,Y 368.931,Z 157.529,A -85,B 0,C 180,E1 -12655.146,E2 -12655.146} C_VEL
LIN {X 0,Y 368.897,Z 157.536,A -85,B 0,C 180,E1 -12659.044,E2 -12659.044} C_VEL
LIN {X 0,Y 368.896,Z 157.57,A -85,B 0,C 180,E1 -12661.064,E2 -12661.064} C_VEL
LIN {X 0,Y 371.41,Z 170.026,A -85,B 0,C 180,E1 -12664.201,E2 -12664.201} C_VEL
LIN {X 0,Y 372.308,Z 175.194,A -85,B 0,C 180,E1 -12665.463,E2 -12665.463} C_VEL
LIN {X 0,Y 371.145,Z 190.013,A -85,B 0,C 180,E1 -12668.824,E2 -12668.824} C_VEL
LIN {X 0,Y 375.816,Z 221.98,A -85,B 0,C 180,E1 -12669.783,E2 -12669.783} C_VEL
LIN {X 0,Y 374.381,Z 298.621,A -85,B 0,C 180,E1 -12671.39,E2 -12671.39} C_VEL
LIN {X 0,Y 373.791,Z 312.23,A -85,B 0,C 180,E1 -12671.891,E2 -12671.891} C_VEL
LIN {X 0,Y 373.081,Z 324.076,A -85,B 0,C 180,E1 -12672.529,E2 -12672.529} C_VEL
LIN {X 0,Y 372.173,Z 336.163,A -85,B 0,C 180,E1 -12673.404,E2 -12673.404} C_VEL
LIN {X 0,Y 371.181,Z 347.718,A -85,B 0,C 180,E1 -12674.488,E2 -12674.488} C_VEL
LIN {X 0,Y 370.384,Z 358.168,A -85,B 0,C 180,E1 -12675.719,E2 -12675.719} C_VEL
LIN {X 0,Y 369.568,Z 367.532,A -85,B 0,C 180,E1 -12677.088,E2 -12677.088} C_VEL
LIN {X 0,Y 368.694,Z 376.612,A -85,B 0,C 180,E1 -12678.733,E2 -12678.733} C_VEL
LIN {X 0,Y 368.14,Z 383.918,A -85,B 0,C 180,E1 -12680.384,E2 -12680.384} C_VEL
LIN {X 0,Y 367.806,Z 388.834,A -85,B 0,C 180,E1 -12681.761,E2 -12681.761} C_VEL
LIN {X 0,Y 367.565,Z 393.595,A -85,B 0,C 180,E1 -12683.412,E2 -12683.412} C_VEL
LIN {X 0,Y 367.442,Z 397.208,A -85,B 0,C 180,E1 -12685.062,E2 -12685.062} C_VEL
LIN {X 0,Y 367.381,Z 399.777,A -85,B 0,C 180,E1 -12686.71,E2 -12686.71} C_VEL
LIN {X 0,Y 367.362,Z 400.967,A -85,B 0,C 180,E1 -12687.807,E2 -12687.807} C_VEL
LIN {X 0,Y 367.419,Z 401.702,A -85,B 0,C 180,E1 -12688.904,E2 -12688.904} C_VEL
LIN {X 0,Y 367.458,Z 402.034,A -85,B 0,C 180,E1 -12690,E2 -12690} C_VEL
LIN {X 0,Y 367.404,Z 401.967,A -85,B 0,C 180,E1 -12691.096,E2 -12691.096} C_VEL
LIN {X 0,Y 367.358,Z 401.494,A -85,B 0,C 180,E1 -12692.193,E2 -12692.193} C_VEL
LIN {X 0,Y 367.377,Z 400.577,A -85,B 0,C 180,E1 -12693.29,E2 -12693.29} C_VEL
LIN {X 0,Y 367.435,Z 399.256,A -85,B 0,C 180,E1 -12694.388,E2 -12694.388} C_VEL
LIN {X 0,Y 367.474,Z 396.532,A -85,B 0,C 180,E1 -12696.004,E2 -12696.004} C_VEL
LIN {X 0,Y 367.745,Z 392.638,A -85,B 0,C 180,E1 -12697.688,E2 -12697.688} C_VEL
LIN {X 0,Y 368.162,Z 387.677,A -85,B 0,C 180,E1 -12699.338,E2 -12699.338} C_VEL
LIN {X 0,Y 368.767,Z 381.436,A -85,B 0,C 180,E1 -12700.986,E2 -12700.986} C_VEL
LIN {X 0,Y 369.649,Z 373.692,A -85,B 0,C 180,E1 -12702.629,E2 -12702.629} C_VEL
LIN {X 0,Y 370.74,Z 363.999,A -85,B 0,C 180,E1 -12704.266,E2 -12704.266} C_VEL
LIN {X 0,Y 371.727,Z 354.032,A -85,B 0,C 180,E1 -12705.629,E2 -12705.629} C_VEL
LIN {X 0,Y 372.79,Z 344.254,A -85,B 0,C 180,E1 -12706.708,E2 -12706.708} C_VEL
LIN {X 0,Y 374.02,Z 331.946,A -85,B 0,C 180,E1 -12707.778,E2 -12707.778} C_VEL
LIN {X 0,Y 375.023,Z 319.993,A -85,B 0,C 180,E1 -12708.577,E2 -12708.577} C_VEL
LIN {X 0,Y 375.888,Z 307.038,A -85,B 0,C 180,E1 -12709.205,E2 -12709.205} C_VEL
LIN {X 0,Y 376.546,Z 293.168,A -85,B 0,C 180,E1 -12709.63,E2 -12709.63} C_VEL
LIN {X 0,Y 377.912,Z 221.198,A -85,B 0,C 180,E1 -12711.169,E2 -12711.169} C_VEL
LIN {X 0,Y 374.244,Z 198.976,A -85,B 0,C 180,E1 -12711.946,E2 -12711.946} C_VEL
LIN {X 0,Y 372.13,Z 188.709,A -85,B 0,C 180,E1 -12712.367,E2 -12712.367} C_VEL
LIN {X 0,Y 373.066,Z 178.217,A -85,B 0,C 180,E1 -12714.753,E2 -12714.753} C_VEL
LIN {X 0,Y 372.325,Z 173.077,A -85,B 0,C 180,E1 -12716.031,E2 -12716.031} C_VEL
LIN {X 0,Y 369.847,Z 161.587,A -85,B 0,C 180,E1 -12719.059,E2 -12719.059} C_VEL
LIN {X 0,Y 368.926,Z 157.54,A -85,B 0,C 180,E1 -12720.2,E2 -12720.2} C_VEL
LIN {X 0,Y 368.894,Z 157.536,A -85,B 0,C 180,E1 -12723.538,E2 -12723.538} C_VEL
LIN {X 0,Y 368.894,Z 157.535,A -85,B 0,C 180,E1 -12726.853,E2 -12726.853} C_VEL
LIN {X 0,Y 368.882,Z 157.538,A -85,B 0,C 180,E1 -12730.373,E2 -12730.373} C_VEL
LIN {X 0,Y 368.876,Z 157.54,A -85,B 0,C 180,E1 -12733.614,E2 -12733.614} C_VEL
LIN {X 0,Y 368.881,Z 157.538,A -85,B 0,C 180,E1 -12736.695,E2 -12736.695} C_VEL
LIN {X 0,Y 368.881,Z 157.533,A -85,B 0,C 180,E1 -12739.647,E2 -12739.647} C_VEL
LIN {X 0,Y 368.891,Z 157.529,A -85,B 0,C 180,E1 -12743.145,E2 -12743.145} C_VEL
LIN {X 0,Y 368.891,Z 157.53,A -85,B 0,C 180,E1 -12746.461,E2 -12746.461} C_VEL
LIN {X 0,Y 368.892,Z 157.53,A -85,B 0,C 180,E1 -12749.042,E2 -12749.042} C_VEL
LIN {X 0,Y 368.902,Z 157.531,A -85,B 0,C 180,E1 -12751.557,E2 -12751.557} C_VEL
LIN {X 0,Y 368.88,Z 157.535,A -85,B 0,C 180,E1 -12755.219,E2 -12755.219} C_VEL
LIN {X 0,Y 368.89,Z 157.525,A -85,B 0,C 180,E1 -12757.602,E2 -12757.602} C_VEL
LIN {X 0,Y 368.893,Z 157.526,A -85,B 0,C 180,E1 -12761.102,E2 -12761.102} C_VEL
LIN {X 0,Y 368.928,Z 157.524,A -85,B 0,C 180,E1 -12764.532,E2 -12764.532} C_VEL
LIN {X 0,Y 369.051,Z 157.513,A -85,B 0,C 180,E1 -12766.79,E2 -12766.79} C_VEL
LIN {X 0,Y 369.051,Z 157.517,A -85,B 0,C 180,E1 -12770.131,E2 -12770.131} C_VEL
LIN {X 0,Y 369.147,Z 157.502,A -85,B 0,C 180,E1 -12773.44,E2 -12773.44} C_VEL
LIN {X 0,Y 369.293,Z 157.482,A -85,B 0,C 180,E1 -12777.818,E2 -12777.818} C_VEL
LIN {X 0,Y 369.293,Z 157.486,A -85,B 0,C 180,E1 -12782.181,E2 -12782.181} C_VEL
LIN {X 0,Y 369.146,Z 157.503,A -85,B 0,C 180,E1 -12786.559,E2 -12786.559} C_VEL
LIN {X 0,Y 369.05,Z 157.518,A -85,B 0,C 180,E1 -12789.868,E2 -12789.868} C_VEL
LIN {X 0,Y 369.03,Z 157.526,A -85,B 0,C 180,E1 -12793.772,E2 -12793.772} C_VEL
LIN {X 0,Y 368.984,Z 157.556,A -85,B 0,C 180,E1 -12797.818,E2 -12797.818} C_VEL
LIN {X 0,Y 371.532,Z 169.191,A -85,B 0,C 180,E1 -12801.063,E2 -12801.063} C_VEL
LIN {X 0,Y 371.988,Z 171.559,A -85,B 0,C 180,E1 -12801.698,E2 -12801.698} C_VEL
LIN {X 0,Y 374.74,Z 179.42,A -85,B 0,C 180,E1 -12802.092,E2 -12802.092} C_VEL
LIN {X 0,Y 378.517,Z 196.843,A -85,B 0,C 180,E1 -12802.775,E2 -12802.775} C_VEL
LIN {X 0,Y 376.57,Z 279.637,A -85,B 0,C 180,E1 -12804.553,E2 -12804.553} C_VEL
LIN {X 0,Y 375.966,Z 292.593,A -85,B 0,C 180,E1 -12805.038,E2 -12805.038} C_VEL
LIN {X 0,Y 375.243,Z 304.985,A -85,B 0,C 180,E1 -12805.716,E2 -12805.716} C_VEL
LIN {X 0,Y 374.365,Z 316.047,A -85,B 0,C 180,E1 -12806.522,E2 -12806.522} C_VEL
LIN {X 0,Y 373.279,Z 327.712,A -85,B 0,C 180,E1 -12807.618,E2 -12807.618} C_VEL
LIN {X 0,Y 372.207,Z 337.653,A -85,B 0,C 180,E1 -12808.782,E2 -12808.782} C_VEL
LIN {X 0,Y 371.161,Z 346.919,A -85,B 0,C 180,E1 -12810.117,E2 -12810.117} C_VEL
LIN {X 0,Y 370.122,Z 355.743,A -85,B 0,C 180,E1 -12811.7,E2 -12811.7} C_VEL
LIN {X 0,Y 369.208,Z 363.769,A -85,B 0,C 180,E1 -12813.505,E2 -12813.505} C_VEL
LIN {X 0,Y 368.653,Z 368.864,A -85,B 0,C 180,E1 -12814.942,E2 -12814.942} C_VEL
LIN {X 0,Y 368.135,Z 373.837,A -85,B 0,C 180,E1 -12816.698,E2 -12816.698} C_VEL
LIN {X 0,Y 367.734,Z 377.468,A -85,B 0,C 180,E1 -12818.412,E2 -12818.412} C_VEL
LIN {X 0,Y 367.398,Z 380.46,A -85,B 0,C 180,E1 -12820.57,E2 -12820.57} C_VEL
LIN {X 0,Y 367.24,Z 381.606,A -85,B 0,C 180,E1 -12822.052,E2 -12822.052} C_VEL
LIN {X 0,Y 367.179,Z 382.006,A -85,B 0,C 180,E1 -12823.555,E2 -12823.555} C_VEL
LIN {X 0,Y 367.211,Z 381.603,A -85,B 0,C 180,E1 -12825.083,E2 -12825.083} C_VEL
LIN {X 0,Y 367.308,Z 380.394,A -85,B 0,C 180,E1 -12826.642,E2 -12826.642} C_VEL
LIN {X 0,Y 367.418,Z 378.279,A -85,B 0,C 180,E1 -12828.244,E2 -12828.244} C_VEL
LIN {X 0,Y 367.673,Z 375.171,A -85,B 0,C 180,E1 -12829.87,E2 -12829.87} C_VEL
LIN {X 0,Y 367.991,Z 370.887,A -85,B 0,C 180,E1 -12831.538,E2 -12831.538} C_VEL
LIN {X 0,Y 368.546,Z 364.244,A -85,B 0,C 180,E1 -12833.507,E2 -12833.507} C_VEL
LIN {X 0,Y 369.152,Z 357.037,A -85,B 0,C 180,E1 -12835.171,E2 -12835.171} C_VEL
LIN {X 0,Y 369.938,Z 348.72,A -85,B 0,C 180,E1 -12836.709,E2 -12836.709} C_VEL
LIN {X 0,Y 370.743,Z 339.552,A -85,B 0,C 180,E1 -12838.092,E2 -12838.092} C_VEL
LIN {X 0,Y 371.553,Z 329.829,A -85,B 0,C 180,E1 -12839.29,E2 -12839.29} C_VEL
LIN {X 0,Y 372.397,Z 319.141,A -85,B 0,C 180,E1 -12840.349,E2 -12840.349} C_VEL
LIN {X 0,Y 373.223,Z 306.835,A -85,B 0,C 180,E1 -12841.304,E2 -12841.304} C_VEL
LIN {X 0,Y 373.929,Z 293.975,A -85,B 0,C 180,E1 -12842.05,E2 -12842.05} C_VEL
LIN {X 0,Y 374.429,Z 280.319,A -85,B 0,C 180,E1 -12842.585,E2 -12842.585} C_VEL
LIN {X 0,Y 374.904,Z 256.63,A -85,B 0,C 180,E1 -12843.113,E2 -12843.113} C_VEL
LIN {X 0,Y 376.002,Z 195.251,A -85,B 0,C 180,E1 -12844.385,E2 -12844.385} C_VEL
LIN {X 0,Y 371.396,Z 170.76,A -85,B 0,C 180,E1 -12845.182,E2 -12845.182} C_VEL
LIN {X 0,Y 369.334,Z 159.538,A -85,B 0,C 180,E1 -12848.219,E2 -12848.219} C_VEL
LIN {X 0,Y 368.935,Z 157.53,A -85,B 0,C 180,E1 -12848.781,E2 -12848.781} C_VEL
LIN {X 0,Y 368.949,Z 157.528,A -85,B 0,C 180,E1 -12852.256,E2 -12852.256} C_VEL
LIN {X 0,Y 369.034,Z 157.518,A -85,B 0,C 180,E1 -12856.228,E2 -12856.228} C_VEL
LIN {X 0,Y 369.054,Z 157.515,A -85,B 0,C 180,E1 -12860.132,E2 -12860.132} C_VEL
LIN {X 0,Y 369.154,Z 157.498,A -85,B 0,C 180,E1 -12863.441,E2 -12863.441} C_VEL
LIN {X 0,Y 369.297,Z 157.483,A -85,B 0,C 180,E1 -12867.819,E2 -12867.819} C_VEL
LIN {X 0,Y 369.292,Z 157.486,A -85,B 0,C 180,E1 -12872.181,E2 -12872.181} C_VEL
LIN {X 0,Y 369.109,Z 157.503,A -85,B 0,C 180,E1 -12875.849,E2 -12875.849} C_VEL
LIN {X 0,Y 368.452,Z 157.586,A -85,B 0,C 180,E1 -12876.76,E2 -12876.76} C_VEL
LIN {X 0,Y 365.567,Z 157.948,A -85,B 0,C 180,E1 -12878.241,E2 -12878.241} C_VEL
LIN {X 0,Y 363.108,Z 158.254,A -85,B 0,C 180,E1 -12879.439,E2 -12879.439} C_VEL
LIN {X 0,Y 362.046,Z 158.386,A -85,B 0,C 180,E1 -12880.366,E2 -12880.366} C_VEL
LIN {X 0,Y 361.957,Z 158.395,A -85,B 0,C 180,E1 -12880.68,E2 -12880.68} C_VEL
LIN {X 0,Y 361.976,Z 158.397,A -85,B 0,C 180,E1 -12883.887,E2 -12883.887} C_VEL
LIN {X 0,Y 361.881,Z 158.406,A -85,B 0,C 180,E1 -12888.103,E2 -12888.103} C_VEL
LIN {X 0,Y 361.849,Z 158.414,A -85,B 0,C 180,E1 -12891.655,E2 -12891.655} C_VEL
LIN {X 0,Y 361.848,Z 158.412,A -85,B 0,C 180,E1 -12895.296,E2 -12895.296} C_VEL
LIN {X 0,Y 361.851,Z 158.41,A -85,B 0,C 180,E1 -12899.074,E2 -12899.074} C_VEL
LIN {X 0,Y 361.843,Z 158.411,A -85,B 0,C 180,E1 -12902.945,E2 -12902.945} C_VEL
LIN {X 0,Y 361.863,Z 158.409,A -85,B 0,C 180,E1 -12905.637,E2 -12905.637} C_VEL
LIN {X 0,Y 361.821,Z 158.416,A -85,B 0,C 180,E1 -12909.018,E2 -12909.018} C_VEL
LIN {X 0,Y 361.824,Z 158.414,A -85,B 0,C 180,E1 -12912.83,E2 -12912.83} C_VEL
LIN {X 0,Y 361.808,Z 158.413,A -85,B 0,C 180,E1 -12915.948,E2 -12915.948} C_VEL
LIN {X 0,Y 361.806,Z 158.417,A -85,B 0,C 180,E1 -12919.249,E2 -12919.249} C_VEL
LIN {X 0,Y 361.855,Z 158.413,A -85,B 0,C 180,E1 -12922.981,E2 -12922.981} C_VEL
LIN {X 0,Y 361.852,Z 158.412,A -85,B 0,C 180,E1 -12926.631,E2 -12926.631} C_VEL
LIN {X 0,Y 361.85,Z 158.408,A -85,B 0,C 180,E1 -12929.67,E2 -12929.67} C_VEL
LIN {X 0,Y 361.849,Z 158.408,A -85,B 0,C 180,E1 -12933.467,E2 -12933.467} C_VEL
LIN {X 0,Y 361.856,Z 158.408,A -85,B 0,C 180,E1 -12937.143,E2 -12937.143} C_VEL
LIN {X 0,Y 361.849,Z 158.412,A -85,B 0,C 180,E1 -12940.721,E2 -12940.721} C_VEL
LIN {X 0,Y 361.89,Z 158.407,A -85,B 0,C 180,E1 -12944.224,E2 -12944.224} C_VEL
LIN {X 0,Y 361.994,Z 158.395,A -85,B 0,C 180,E1 -12946.528,E2 -12946.528} C_VEL
LIN {X 0,Y 361.989,Z 158.393,A -85,B 0,C 180,E1 -12949.937,E2 -12949.937} C_VEL
LIN {X 0,Y 362.113,Z 158.375,A -85,B 0,C 180,E1 -12953.313,E2 -12953.313} C_VEL
LIN {X 0,Y 362.253,Z 158.361,A -85,B 0,C 180,E1 -12957.777,E2 -12957.777} C_VEL
LIN {X 0,Y 362.168,Z 158.368,A -85,B 0,C 180,E1 -12961.112,E2 -12961.112} C_VEL
LIN {X 0,Y 362.252,Z 158.362,A -85,B 0,C 180,E1 -12962.224,E2 -12962.224} C_VEL
LIN {X 0,Y 362.113,Z 158.375,A -85,B 0,C 180,E1 -12966.688,E2 -12966.688} C_VEL
